LIN {X 0,Y 573.015,Z 252.998,A -85,B 0,C 180,E1 -2072.459,E2 -2072.459} C_VEL
LIN {X 0,Y 573.012,Z 250.251,A -85,B 0,C 180,E1 -2073.163,E2 -2073.163} C_VEL
LIN {X 0,Y 573.036,Z 245.506,A -85,B 0,C 180,E1 -2074.043,E2 -2074.043} C_VEL
LIN {X 0,Y 573.097,Z 240.544,A -85,B 0,C 180,E1 -2074.747,E2 -2074.747} C_VEL
LIN {X 0,Y 573.027,Z 234.186,A -85,B 0,C 180,E1 -2075.453,E2 -2075.453} C_VEL
LIN {X 0,Y 573.106,Z 227.017,A -85,B 0,C 180,E1 -2076.07,E2 -2076.07} C_VEL
LIN {X 0,Y 573.128,Z 220.284,A -85,B 0,C 180,E1 -2076.527,E2 -2076.527} C_VEL
LIN {X 0,Y 573.236,Z 211.927,A -85,B 0,C 180,E1 -2076.962,E2 -2076.962} C_VEL
LIN {X 0,Y 573.056,Z 204.686,A -85,B 0,C 180,E1 -2077.243,E2 -2077.243} C_VEL
LIN {X 0,Y 572.921,Z 203.423,A -85,B 0,C 180,E1 -2077.311,E2 -2077.311} C_VEL
LIN {X 0,Y 572.967,Z 198.327,A -85,B 0,C 180,E1 -2080.601,E2 -2080.601} C_VEL
LIN {X 0,Y 572.969,Z 193.92,A -85,B 0,C 180,E1 -2083.476,E2 -2083.476} C_VEL
LIN {X 0,Y 572.966,Z 189.58,A -85,B 0,C 180,E1 -2086.386,E2 -2086.386} C_VEL
LIN {X 0,Y 572.998,Z 185.595,A -85,B 0,C 180,E1 -2089.338,E2 -2089.338} C_VEL
LIN {X 0,Y 573.019,Z 182.564,A -85,B 0,C 180,E1 -2091.588,E2 -2091.588} C_VEL
LIN {X 0,Y 573.073,Z 179.507,A -85,B 0,C 180,E1 -2093.871,E2 -2093.871} C_VEL
LIN {X 0,Y 573.141,Z 176.057,A -85,B 0,C 180,E1 -2096.472,E2 -2096.472} C_VEL
LIN {X 0,Y 573.16,Z 173.251,A -85,B 0,C 180,E1 -2098.567,E2 -2098.567} C_VEL
LIN {X 0,Y 573.151,Z 172.095,A -85,B 0,C 180,E1 -2099.471,E2 -2099.471} C_VEL
LIN {X 0,Y 573.245,Z 172.076,A -85,B 0,C 180,E1 -2102.227,E2 -2102.227} C_VEL
LIN {X 0,Y 573.233,Z 172.077,A -85,B 0,C 180,E1 -2104.771,E2 -2104.771} C_VEL
LIN {X 0,Y 573.247,Z 172.08,A -85,B 0,C 180,E1 -2107.165,E2 -2107.165} C_VEL
LIN {X 0,Y 573.241,Z 172.079,A -85,B 0,C 180,E1 -2109.606,E2 -2109.606} C_VEL
LIN {X 0,Y 573.237,Z 172.078,A -85,B 0,C 180,E1 -2112.641,E2 -2112.641} C_VEL
LIN {X 0,Y 573.229,Z 172.077,A -85,B 0,C 180,E1 -2115.666,E2 -2115.666} C_VEL
LIN {X 0,Y 573.238,Z 172.08,A -85,B 0,C 180,E1 -2118.543,E2 -2118.543} C_VEL
LIN {X 0,Y 573.242,Z 172.076,A -85,B 0,C 180,E1 -2121.298,E2 -2121.298} C_VEL
LIN {X 0,Y 573.257,Z 172.074,A -85,B 0,C 180,E1 -2124.01,E2 -2124.01} C_VEL
LIN {X 0,Y 573.276,Z 172.079,A -85,B 0,C 180,E1 -2126.518,E2 -2126.518} C_VEL
LIN {X 0,Y 573.236,Z 172.076,A -85,B 0,C 180,E1 -2129.114,E2 -2129.114} C_VEL
LIN {X 0,Y 573.256,Z 172.077,A -85,B 0,C 180,E1 -2131.967,E2 -2131.967} C_VEL
LIN {X 0,Y 573.249,Z 172.075,A -85,B 0,C 180,E1 -2134.59,E2 -2134.59} C_VEL
LIN {X 0,Y 573.23,Z 172.08,A -85,B 0,C 180,E1 -2137.662,E2 -2137.662} C_VEL
LIN {X 0,Y 573.248,Z 172.082,A -85,B 0,C 180,E1 -2139.923,E2 -2139.923} C_VEL
LIN {X 0,Y 573.253,Z 172.074,A -85,B 0,C 180,E1 -2142.988,E2 -2142.988} C_VEL
LIN {X 0,Y 573.263,Z 172.078,A -85,B 0,C 180,E1 -2145.807,E2 -2145.807} C_VEL
LIN {X 0,Y 573.272,Z 172.071,A -85,B 0,C 180,E1 -2148.734,E2 -2148.734} C_VEL
LIN {X 0,Y 573.296,Z 172.074,A -85,B 0,C 180,E1 -2151.541,E2 -2151.541} C_VEL
LIN {X 0,Y 573.283,Z 172.069,A -85,B 0,C 180,E1 -2154.372,E2 -2154.372} C_VEL
LIN {X 0,Y 573.296,Z 172.076,A -85,B 0,C 180,E1 -2157.189,E2 -2157.189} C_VEL
LIN {X 0,Y 573.3,Z 172.066,A -85,B 0,C 180,E1 -2160,E2 -2160} C_VEL
LIN {X 0,Y 573.3,Z 172.076,A -85,B 0,C 180,E1 -2162.811,E2 -2162.811} C_VEL
LIN {X 0,Y 573.265,Z 172.071,A -85,B 0,C 180,E1 -2165.628,E2 -2165.628} C_VEL
LIN {X 0,Y 573.274,Z 172.078,A -85,B 0,C 180,E1 -2168.46,E2 -2168.46} C_VEL
LIN {X 0,Y 573.259,Z 172.073,A -85,B 0,C 180,E1 -2171.312,E2 -2171.312} C_VEL
LIN {X 0,Y 573.268,Z 172.079,A -85,B 0,C 180,E1 -2174.424,E2 -2174.424} C_VEL
LIN {X 0,Y 573.233,Z 172.075,A -85,B 0,C 180,E1 -2177.112,E2 -2177.112} C_VEL
LIN {X 0,Y 573.22,Z 172.087,A -85,B 0,C 180,E1 -2180.078,E2 -2180.078} C_VEL
LIN {X 0,Y 573.204,Z 172.083,A -85,B 0,C 180,E1 -2182.339,E2 -2182.339} C_VEL
LIN {X 0,Y 573.212,Z 172.082,A -85,B 0,C 180,E1 -2185.412,E2 -2185.412} C_VEL
LIN {X 0,Y 573.166,Z 172.084,A -85,B 0,C 180,E1 -2188.568,E2 -2188.568} C_VEL
LIN {X 0,Y 573.204,Z 172.081,A -85,B 0,C 180,E1 -2190.995,E2 -2190.995} C_VEL
LIN {X 0,Y 573.253,Z 172.081,A -85,B 0,C 180,E1 -2193.525,E2 -2193.525} C_VEL
LIN {X 0,Y 573.177,Z 172.084,A -85,B 0,C 180,E1 -2196.054,E2 -2196.054} C_VEL
LIN {X 0,Y 573.225,Z 172.08,A -85,B 0,C 180,E1 -2198.703,E2 -2198.703} C_VEL
LIN {X 0,Y 573.205,Z 172.082,A -85,B 0,C 180,E1 -2201.592,E2 -2201.592} C_VEL
LIN {X 0,Y 573.214,Z 172.08,A -85,B 0,C 180,E1 -2204.336,E2 -2204.336} C_VEL
LIN {X 0,Y 573.233,Z 172.076,A -85,B 0,C 180,E1 -2207.36,E2 -2207.36} C_VEL
LIN {X 0,Y 573.239,Z 172.081,A -85,B 0,C 180,E1 -2210.394,E2 -2210.394} C_VEL
LIN {X 0,Y 573.247,Z 172.077,A -85,B 0,C 180,E1 -2213.079,E2 -2213.079} C_VEL
LIN {X 0,Y 573.262,Z 172.073,A -85,B 0,C 180,E1 -2215.672,E2 -2215.672} C_VEL
LIN {X 0,Y 573.241,Z 172.084,A -85,B 0,C 180,E1 -2218.186,E2 -2218.186} C_VEL
LIN {X 0,Y 573.246,Z 172.092,A -85,B 0,C 180,E1 -2219.909,E2 -2219.909} C_VEL
LIN {X 0,Y 574.683,Z 179.226,A -85,B 0,C 180,E1 -2221.116,E2 -2221.116} C_VEL
LIN {X 0,Y 574.417,Z 195.626,A -85,B 0,C 180,E1 -2223.566,E2 -2223.566} C_VEL
LIN {X 0,Y 574.13,Z 214.897,A -85,B 0,C 180,E1 -2226.339,E2 -2226.339} C_VEL
LIN {X 0,Y 573.948,Z 232.888,A -85,B 0,C 180,E1 -2228.868,E2 -2228.868} C_VEL
LIN {X 0,Y 573.731,Z 253.864,A -85,B 0,C 180,E1 -2231.799,E2 -2231.799} C_VEL
LIN {X 0,Y 573.504,Z 273.808,A -85,B 0,C 180,E1 -2234.543,E2 -2234.543} C_VEL
LIN {X 0,Y 573.35,Z 293.752,A -85,B 0,C 180,E1 -2237.254,E2 -2237.254} C_VEL
LIN {X 0,Y 573.34,Z 295.393,A -85,B 0,C 180,E1 -2237.434,E2 -2237.434} C_VEL
LIN {X 0,Y 573.925,Z 301.68,A -85,B 0,C 180,E1 -2237.537,E2 -2237.537} C_VEL
LIN {X 0,Y 573.782,Z 314.725,A -85,B 0,C 180,E1 -2237.826,E2 -2237.826} C_VEL
LIN {X 0,Y 573.709,Z 327.272,A -85,B 0,C 180,E1 -2238.25,E2 -2238.25} C_VEL
LIN {X 0,Y 573.61,Z 338.953,A -85,B 0,C 180,E1 -2238.785,E2 -2238.785} C_VEL
LIN {X 0,Y 573.478,Z 349.603,A -85,B 0,C 180,E1 -2239.408,E2 -2239.408} C_VEL
LIN {X 0,Y 573.362,Z 360.484,A -85,B 0,C 180,E1 -2240.209,E2 -2240.209} C_VEL
LIN {X 0,Y 573.24,Z 371.123,A -85,B 0,C 180,E1 -2241.186,E2 -2241.186} C_VEL
LIN {X 0,Y 573.16,Z 378.968,A -85,B 0,C 180,E1 -2242.072,E2 -2242.072} C_VEL
LIN {X 0,Y 573.073,Z 386.586,A -85,B 0,C 180,E1 -2243.127,E2 -2243.127} C_VEL
LIN {X 0,Y 573.07,Z 393.684,A -85,B 0,C 180,E1 -2244.371,E2 -2244.371} C_VEL
LIN {X 0,Y 573.028,Z 398.375,A -85,B 0,C 180,E1 -2245.428,E2 -2245.428} C_VEL
LIN {X 0,Y 573.022,Z 401.962,A -85,B 0,C 180,E1 -2246.485,E2 -2246.485} C_VEL
LIN {X 0,Y 572.959,Z 403.812,A -85,B 0,C 180,E1 -2247.189,E2 -2247.189} C_VEL
LIN {X 0,Y 572.94,Z 405.201,A -85,B 0,C 180,E1 -2247.892,E2 -2247.892} C_VEL
LIN {X 0,Y 572.94,Z 406.786,A -85,B 0,C 180,E1 -2249.298,E2 -2249.298} C_VEL
LIN {X 0,Y 572.938,Z 407,A -85,B 0,C 180,E1 -2250.001,E2 -2250.001} C_VEL
LIN {X 0,Y 572.946,Z 406.185,A -85,B 0,C 180,E1 -2251.407,E2 -2251.407} C_VEL
LIN {X 0,Y 572.94,Z 405.197,A -85,B 0,C 180,E1 -2252.11,E2 -2252.11} C_VEL
LIN {X 0,Y 572.959,Z 403.806,A -85,B 0,C 180,E1 -2252.813,E2 -2252.813} C_VEL
LIN {X 0,Y 573.015,Z 400.893,A -85,B 0,C 180,E1 -2253.869,E2 -2253.869} C_VEL
LIN {X 0,Y 572.963,Z 396.946,A -85,B 0,C 180,E1 -2254.926,E2 -2254.926} C_VEL
LIN {X 0,Y 573.065,Z 390.872,A -85,B 0,C 180,E1 -2256.161,E2 -2256.161} C_VEL
LIN {X 0,Y 573.12,Z 384.232,A -85,B 0,C 180,E1 -2257.222,E2 -2257.222} C_VEL
LIN {X 0,Y 573.199,Z 375.984,A -85,B 0,C 180,E1 -2258.284,E2 -2258.284} C_VEL
LIN {X 0,Y 573.287,Z 367.53,A -85,B 0,C 180,E1 -2259.171,E2 -2259.171} C_VEL
LIN {X 0,Y 573.426,Z 357.088,A -85,B 0,C 180,E1 -2260.059,E2 -2260.059} C_VEL
LIN {X 0,Y 573.537,Z 345.389,A -85,B 0,C 180,E1 -2260.856,E2 -2260.856} C_VEL
LIN {X 0,Y 573.654,Z 334.274,A -85,B 0,C 180,E1 -2261.448,E2 -2261.448} C_VEL
LIN {X 0,Y 573.759,Z 321.154,A -85,B 0,C 180,E1 -2261.975,E2 -2261.975} C_VEL
LIN {X 0,Y 573.845,Z 308.489,A -85,B 0,C 180,E1 -2262.332,E2 -2262.332} C_VEL
LIN {X 0,Y 573.821,Z 298.547,A -85,B 0,C 180,E1 -2262.512,E2 -2262.512} C_VEL
LIN {X 0,Y 573.297,Z 294.902,A -85,B 0,C 180,E1 -2262.591,E2 -2262.591} C_VEL
LIN {X 0,Y 573.449,Z 276.454,A -85,B 0,C 180,E1 -2265.097,E2 -2265.097} C_VEL
LIN {X 0,Y 573.671,Z 256.51,A -85,B 0,C 180,E1 -2267.836,E2 -2267.836} C_VEL
LIN {X 0,Y 573.902,Z 236.566,A -85,B 0,C 180,E1 -2270.615,E2 -2270.615} C_VEL
LIN {X 0,Y 574.126,Z 217.882,A -85,B 0,C 180,E1 -2273.24,E2 -2273.24} C_VEL
LIN {X 0,Y 574.361,Z 197.613,A -85,B 0,C 180,E1 -2276.137,E2 -2276.137} C_VEL
LIN {X 0,Y 574.695,Z 180.513,A -85,B 0,C 180,E1 -2278.686,E2 -2278.686} C_VEL
LIN {X 0,Y 574.272,Z 176.66,A -85,B 0,C 180,E1 -2279.31,E2 -2279.31} C_VEL
LIN {X 0,Y 573.228,Z 172.084,A -85,B 0,C 180,E1 -2280.094,E2 -2280.094} C_VEL
LIN {X 0,Y 573.226,Z 172.082,A -85,B 0,C 180,E1 -2282.648,E2 -2282.648} C_VEL
LIN {X 0,Y 573.191,Z 172.089,A -85,B 0,C 180,E1 -2285.19,E2 -2285.19} C_VEL
LIN {X 0,Y 573.231,Z 172.079,A -85,B 0,C 180,E1 -2287.809,E2 -2287.809} C_VEL
LIN {X 0,Y 573.25,Z 172.08,A -85,B 0,C 180,E1 -2290.525,E2 -2290.525} C_VEL
LIN {X 0,Y 573.241,Z 172.078,A -85,B 0,C 180,E1 -2293.36,E2 -2293.36} C_VEL
LIN {X 0,Y 573.241,Z 172.077,A -85,B 0,C 180,E1 -2296.641,E2 -2296.641} C_VEL
LIN {X 0,Y 573.25,Z 172.08,A -85,B 0,C 180,E1 -2299.475,E2 -2299.475} C_VEL
LIN {X 0,Y 573.229,Z 172.08,A -85,B 0,C 180,E1 -2302.192,E2 -2302.192} C_VEL
LIN {X 0,Y 573.205,Z 172.084,A -85,B 0,C 180,E1 -2305.234,E2 -2305.234} C_VEL
LIN {X 0,Y 573.152,Z 172.129,A -85,B 0,C 180,E1 -2306.088,E2 -2306.088} C_VEL
LIN {X 0,Y 573.182,Z 181.357,A -85,B 0,C 180,E1 -2308.593,E2 -2308.593} C_VEL
LIN {X 0,Y 573.206,Z 191.116,A -85,B 0,C 180,E1 -2311.434,E2 -2311.434} C_VEL
LIN {X 0,Y 573.264,Z 200.054,A -85,B 0,C 180,E1 -2314.201,E2 -2314.201} C_VEL
LIN {X 0,Y 573.203,Z 208.222,A -85,B 0,C 180,E1 -2316.899,E2 -2316.899} C_VEL
LIN {X 0,Y 573.192,Z 215.13,A -85,B 0,C 180,E1 -2319.171,E2 -2319.171} C_VEL
LIN {X 0,Y 573.142,Z 222.895,A -85,B 0,C 180,E1 -2321.779,E2 -2321.779} C_VEL
LIN {X 0,Y 573.106,Z 230.685,A -85,B 0,C 180,E1 -2324.348,E2 -2324.348} C_VEL
LIN {X 0,Y 573.075,Z 239.587,A -85,B 0,C 180,E1 -2327.247,E2 -2327.247} C_VEL
LIN {X 0,Y 573.088,Z 240.711,A -85,B 0,C 180,E1 -2327.551,E2 -2327.551} C_VEL
LIN {X 0,Y 573.868,Z 246.446,A -85,B 0,C 180,E1 -2327.669,E2 -2327.669} C_VEL
LIN {X 0,Y 573.774,Z 259.872,A -85,B 0,C 180,E1 -2328.026,E2 -2328.026} C_VEL
LIN {X 0,Y 573.64,Z 271.829,A -85,B 0,C 180,E1 -2328.485,E2 -2328.485} C_VEL
LIN {X 0,Y 573.551,Z 283.172,A -85,B 0,C 180,E1 -2329.061,E2 -2329.061} C_VEL
LIN {X 0,Y 573.454,Z 294.108,A -85,B 0,C 180,E1 -2329.764,E2 -2329.764} C_VEL
LIN {X 0,Y 573.34,Z 303.126,A -85,B 0,C 180,E1 -2330.475,E2 -2330.475} C_VEL
LIN {X 0,Y 573.244,Z 312.371,A -85,B 0,C 180,E1 -2331.362,E2 -2331.362} C_VEL
LIN {X 0,Y 573.143,Z 321.354,A -85,B 0,C 180,E1 -2332.425,E2 -2332.425} C_VEL
LIN {X 0,Y 573.091,Z 327.919,A -85,B 0,C 180,E1 -2333.382,E2 -2333.382} C_VEL
LIN {X 0,Y 573.071,Z 333.463,A -85,B 0,C 180,E1 -2334.37,E2 -2334.37} C_VEL
LIN {X 0,Y 573.029,Z 338.204,A -85,B 0,C 180,E1 -2335.428,E2 -2335.428} C_VEL
LIN {X 0,Y 573.022,Z 341.832,A -85,B 0,C 180,E1 -2336.484,E2 -2336.484} C_VEL
LIN {X 0,Y 572.959,Z 343.69,A -85,B 0,C 180,E1 -2337.188,E2 -2337.188} C_VEL
LIN {X 0,Y 572.938,Z 345.134,A -85,B 0,C 180,E1 -2337.891,E2 -2337.891} C_VEL
LIN {X 0,Y 572.942,Z 346.754,A -85,B 0,C 180,E1 -2339.297,E2 -2339.297} C_VEL
LIN {X 0,Y 572.938,Z 346.996,A -85,B 0,C 180,E1 -2340,E2 -2340} C_VEL
LIN {X 0,Y 572.941,Z 346.813,A -85,B 0,C 180,E1 -2340.703,E2 -2340.703} C_VEL
LIN {X 0,Y 572.937,Z 345.275,A -85,B 0,C 180,E1 -2342.109,E2 -2342.109} C_VEL
LIN {X 0,Y 572.96,Z 343.908,A -85,B 0,C 180,E1 -2342.812,E2 -2342.812} C_VEL
LIN {X 0,Y 573.015,Z 341.039,A -85,B 0,C 180,E1 -2343.868,E2 -2343.868} C_VEL
LIN {X 0,Y 572.963,Z 337.14,A -85,B 0,C 180,E1 -2344.926,E2 -2344.926} C_VEL
LIN {X 0,Y 573.075,Z 332.097,A -85,B 0,C 180,E1 -2345.984,E2 -2345.984} C_VEL
LIN {X 0,Y 573.084,Z 325.762,A -85,B 0,C 180,E1 -2347.044,E2 -2347.044} C_VEL
LIN {X 0,Y 573.175,Z 317.867,A -85,B 0,C 180,E1 -2348.106,E2 -2348.106} C_VEL
LIN {X 0,Y 573.254,Z 309.793,A -85,B 0,C 180,E1 -2348.993,E2 -2348.993} C_VEL
LIN {X 0,Y 573.336,Z 299.936,A -85,B 0,C 180,E1 -2349.882,E2 -2349.882} C_VEL
LIN {X 0,Y 573.464,Z 288.94,A -85,B 0,C 180,E1 -2350.679,E2 -2350.679} C_VEL
LIN {X 0,Y 573.587,Z 276.923,A -85,B 0,C 180,E1 -2351.364,E2 -2351.364} C_VEL
LIN {X 0,Y 573.702,Z 264.987,A -85,B 0,C 180,E1 -2351.886,E2 -2351.886} C_VEL
LIN {X 0,Y 573.833,Z 251.33,A -85,B 0,C 180,E1 -2352.309,E2 -2352.309} C_VEL
LIN {X 0,Y 573.604,Z 244.173,A -85,B 0,C 180,E1 -2352.471,E2 -2352.471} C_VEL
LIN {X 0,Y 573.043,Z 240.491,A -85,B 0,C 180,E1 -2352.551,E2 -2352.551} C_VEL
LIN {X 0,Y 573.085,Z 230.959,A -85,B 0,C 180,E1 -2355.652,E2 -2355.652} C_VEL
LIN {X 0,Y 573.102,Z 223.166,A -85,B 0,C 180,E1 -2358.223,E2 -2358.223} C_VEL
LIN {X 0,Y 573.143,Z 221.241,A -85,B 0,C 180,E1 -2358.862,E2 -2358.862} C_VEL
LIN {X 0,Y 572.509,Z 219.635,A -85,B 0,C 180,E1 -2359.426,E2 -2359.426} C_VEL
LIN {X 0,Y 569.679,Z 217.271,A -85,B 0,C 180,E1 -2360.35,E2 -2360.35} C_VEL
LIN {X 0,Y 567.27,Z 215.411,A -85,B 0,C 180,E1 -2361.093,E2 -2361.093} C_VEL
LIN {X 0,Y 566.231,Z 213.9,A -85,B 0,C 180,E1 -2361.665,E2 -2361.665} C_VEL
LIN {X 0,Y 566.145,Z 213.329,A -85,B 0,C 180,E1 -2361.857,E2 -2361.857} C_VEL
LIN {X 0,Y 566.188,Z 205.251,A -85,B 0,C 180,E1 -2364.572,E2 -2364.572} C_VEL
LIN {X 0,Y 566.243,Z 197.135,A -85,B 0,C 180,E1 -2367.338,E2 -2367.338} C_VEL
LIN {X 0,Y 566.283,Z 189.921,A -85,B 0,C 180,E1 -2369.764,E2 -2369.764} C_VEL
LIN {X 0,Y 566.353,Z 182.564,A -85,B 0,C 180,E1 -2372.249,E2 -2372.249} C_VEL
LIN {X 0,Y 566.349,Z 174.409,A -85,B 0,C 180,E1 -2375.013,E2 -2375.013} C_VEL
LIN {X 0,Y 566.156,Z 172.965,A -85,B 0,C 180,E1 -2375.555,E2 -2375.555} C_VEL
LIN {X 0,Y 566.211,Z 172.954,A -85,B 0,C 180,E1 -2378.557,E2 -2378.557} C_VEL
LIN {X 0,Y 566.177,Z 172.964,A -85,B 0,C 180,E1 -2381.14,E2 -2381.14} C_VEL
LIN {X 0,Y 566.162,Z 172.961,A -85,B 0,C 180,E1 -2383.947,E2 -2383.947} C_VEL
LIN {X 0,Y 566.205,Z 172.955,A -85,B 0,C 180,E1 -2386.945,E2 -2386.945} C_VEL
LIN {X 0,Y 566.212,Z 172.953,A -85,B 0,C 180,E1 -2389.801,E2 -2389.801} C_VEL
LIN {X 0,Y 566.191,Z 172.959,A -85,B 0,C 180,E1 -2392.601,E2 -2392.601} C_VEL
LIN {X 0,Y 566.189,Z 172.959,A -85,B 0,C 180,E1 -2395.18,E2 -2395.18} C_VEL
LIN {X 0,Y 566.235,Z 172.951,A -85,B 0,C 180,E1 -2397.743,E2 -2397.743} C_VEL
LIN {X 0,Y 566.122,Z 172.971,A -85,B 0,C 180,E1 -2400.343,E2 -2400.343} C_VEL
LIN {X 0,Y 566.099,Z 173.398,A -85,B 0,C 180,E1 -2401.041,E2 -2401.041} C_VEL
LIN {X 0,Y 566.102,Z 176.607,A -85,B 0,C 180,E1 -2403.452,E2 -2403.452} C_VEL
LIN {X 0,Y 566.036,Z 179.691,A -85,B 0,C 180,E1 -2405.811,E2 -2405.811} C_VEL
LIN {X 0,Y 565.978,Z 183.82,A -85,B 0,C 180,E1 -2408.893,E2 -2408.893} C_VEL
LIN {X 0,Y 565.914,Z 187.813,A -85,B 0,C 180,E1 -2411.912,E2 -2411.912} C_VEL
LIN {X 0,Y 565.885,Z 190.906,A -85,B 0,C 180,E1 -2414.143,E2 -2414.143} C_VEL
LIN {X 0,Y 565.881,Z 193.87,A -85,B 0,C 180,E1 -2416.35,E2 -2416.35} C_VEL
LIN {X 0,Y 565.884,Z 198.186,A -85,B 0,C 180,E1 -2419.263,E2 -2419.263} C_VEL
LIN {X 0,Y 565.857,Z 203.453,A -85,B 0,C 180,E1 -2422.708,E2 -2422.708} C_VEL
LIN {X 0,Y 566.167,Z 211.205,A -85,B 0,C 180,E1 -2423.01,E2 -2423.01} C_VEL
LIN {X 0,Y 566.114,Z 218.9,A -85,B 0,C 180,E1 -2423.401,E2 -2423.401} C_VEL
LIN {X 0,Y 566.062,Z 225.793,A -85,B 0,C 180,E1 -2423.852,E2 -2423.852} C_VEL
LIN {X 0,Y 565.983,Z 231.354,A -85,B 0,C 180,E1 -2424.298,E2 -2424.298} C_VEL
LIN {X 0,Y 566.01,Z 238.313,A -85,B 0,C 180,E1 -2425.013,E2 -2425.013} C_VEL
LIN {X 0,Y 565.97,Z 243.753,A -85,B 0,C 180,E1 -2425.726,E2 -2425.726} C_VEL
LIN {X 0,Y 565.969,Z 248.043,A -85,B 0,C 180,E1 -2426.439,E2 -2426.439} C_VEL
LIN {X 0,Y 565.892,Z 251.374,A -85,B 0,C 180,E1 -2427.152,E2 -2427.152} C_VEL
LIN {X 0,Y 565.855,Z 253.859,A -85,B 0,C 180,E1 -2427.864,E2 -2427.864} C_VEL
LIN {X 0,Y 565.847,Z 255.567,A -85,B 0,C 180,E1 -2428.576,E2 -2428.576} C_VEL
LIN {X 0,Y 565.841,Z 256.57,A -85,B 0,C 180,E1 -2429.287,E2 -2429.287} C_VEL
LIN {X 0,Y 565.839,Z 256.937,A -85,B 0,C 180,E1 -2429.999,E2 -2429.999} C_VEL
LIN {X 0,Y 565.841,Z 256.676,A -85,B 0,C 180,E1 -2430.711,E2 -2430.711} C_VEL
LIN {X 0,Y 565.848,Z 255.761,A -85,B 0,C 180,E1 -2431.422,E2 -2431.422} C_VEL
LIN {X 0,Y 565.854,Z 254.12,A -85,B 0,C 180,E1 -2432.134,E2 -2432.134} C_VEL
LIN {X 0,Y 565.935,Z 250.247,A -85,B 0,C 180,E1 -2433.203,E2 -2433.203} C_VEL
LIN {X 0,Y 565.952,Z 245.495,A -85,B 0,C 180,E1 -2434.094,E2 -2434.094} C_VEL
LIN {X 0,Y 566.024,Z 240.534,A -85,B 0,C 180,E1 -2434.807,E2 -2434.807} C_VEL
LIN {X 0,Y 565.954,Z 234.166,A -85,B 0,C 180,E1 -2435.522,E2 -2435.522} C_VEL
LIN {X 0,Y 566.045,Z 228.167,A -85,B 0,C 180,E1 -2436.057,E2 -2436.057} C_VEL
LIN {X 0,Y 566.071,Z 220.396,A -85,B 0,C 180,E1 -2436.601,E2 -2436.601} C_VEL
LIN {X 0,Y 566.152,Z 214.044,A -85,B 0,C 180,E1 -2436.953,E2 -2436.953} C_VEL
LIN {X 0,Y 566.153,Z 206.734,A -85,B 0,C 180,E1 -2437.264,E2 -2437.264} C_VEL
LIN {X 0,Y 565.854,Z 203.456,A -85,B 0,C 180,E1 -2437.38,E2 -2437.38} C_VEL
LIN {X 0,Y 565.879,Z 198.326,A -85,B 0,C 180,E1 -2440.736,E2 -2440.736} C_VEL
LIN {X 0,Y 565.871,Z 193.997,A -85,B 0,C 180,E1 -2443.648,E2 -2443.648} C_VEL
LIN {X 0,Y 565.916,Z 190.002,A -85,B 0,C 180,E1 -2446.596,E2 -2446.596} C_VEL
LIN {X 0,Y 565.936,Z 185.968,A -85,B 0,C 180,E1 -2449.589,E2 -2449.589} C_VEL
LIN {X 0,Y 565.963,Z 182.909,A -85,B 0,C 180,E1 -2451.871,E2 -2451.871} C_VEL
LIN {X 0,Y 566.03,Z 179.83,A -85,B 0,C 180,E1 -2454.187,E2 -2454.187} C_VEL
LIN {X 0,Y 566.079,Z 176.631,A -85,B 0,C 180,E1 -2456.633,E2 -2456.633} C_VEL
LIN {X 0,Y 566.102,Z 173.527,A -85,B 0,C 180,E1 -2458.957,E2 -2458.957} C_VEL
LIN {X 0,Y 566.126,Z 172.97,A -85,B 0,C 180,E1 -2459.772,E2 -2459.772} C_VEL
LIN {X 0,Y 566.198,Z 172.953,A -85,B 0,C 180,E1 -2462.428,E2 -2462.428} C_VEL
LIN {X 0,Y 566.195,Z 172.955,A -85,B 0,C 180,E1 -2464.991,E2 -2464.991} C_VEL
LIN {X 0,Y 566.191,Z 172.961,A -85,B 0,C 180,E1 -2467.46,E2 -2467.46} C_VEL
LIN {X 0,Y 566.212,Z 172.95,A -85,B 0,C 180,E1 -2470.197,E2 -2470.197} C_VEL
LIN {X 0,Y 566.199,Z 172.96,A -85,B 0,C 180,E1 -2473.053,E2 -2473.053} C_VEL
LIN {X 0,Y 566.193,Z 172.953,A -85,B 0,C 180,E1 -2476.047,E2 -2476.047} C_VEL
LIN {X 0,Y 566.205,Z 172.96,A -85,B 0,C 180,E1 -2478.863,E2 -2478.863} C_VEL
LIN {X 0,Y 566.182,Z 172.954,A -85,B 0,C 180,E1 -2481.636,E2 -2481.636} C_VEL
LIN {X 0,Y 566.205,Z 172.956,A -85,B 0,C 180,E1 -2484.311,E2 -2484.311} C_VEL
LIN {X 0,Y 566.221,Z 172.952,A -85,B 0,C 180,E1 -2486.898,E2 -2486.898} C_VEL
LIN {X 0,Y 566.185,Z 172.953,A -85,B 0,C 180,E1 -2489.407,E2 -2489.407} C_VEL
LIN {X 0,Y 566.219,Z 172.952,A -85,B 0,C 180,E1 -2491.858,E2 -2491.858} C_VEL
LIN {X 0,Y 566.217,Z 172.956,A -85,B 0,C 180,E1 -2494.251,E2 -2494.251} C_VEL
LIN {X 0,Y 566.183,Z 172.955,A -85,B 0,C 180,E1 -2496.713,E2 -2496.713} C_VEL
LIN {X 0,Y 566.21,Z 172.955,A -85,B 0,C 180,E1 -2499.663,E2 -2499.663} C_VEL
LIN {X 0,Y 566.194,Z 172.953,A -85,B 0,C 180,E1 -2502.668,E2 -2502.668} C_VEL
LIN {X 0,Y 566.223,Z 172.956,A -85,B 0,C 180,E1 -2505.626,E2 -2505.626} C_VEL
LIN {X 0,Y 566.264,Z 172.944,A -85,B 0,C 180,E1 -2508.654,E2 -2508.654} C_VEL
LIN {X 0,Y 566.238,Z 172.955,A -85,B 0,C 180,E1 -2511.434,E2 -2511.434} C_VEL
LIN {X 0,Y 566.249,Z 172.945,A -85,B 0,C 180,E1 -2514.302,E2 -2514.302} C_VEL
LIN {X 0,Y 566.26,Z 172.944,A -85,B 0,C 180,E1 -2517.866,E2 -2517.866} C_VEL
LIN {X 0,Y 566.299,Z 172.943,A -85,B 0,C 180,E1 -2520.711,E2 -2520.711} C_VEL
LIN {X 0,Y 566.265,Z 172.953,A -85,B 0,C 180,E1 -2522.846,E2 -2522.846} C_VEL
LIN {X 0,Y 566.234,Z 172.947,A -85,B 0,C 180,E1 -2525.699,E2 -2525.699} C_VEL
LIN {X 0,Y 566.217,Z 172.958,A -85,B 0,C 180,E1 -2528.566,E2 -2528.566} C_VEL
LIN {X 0,Y 566.229,Z 172.948,A -85,B 0,C 180,E1 -2531.455,E2 -2531.455} C_VEL
LIN {X 0,Y 566.221,Z 172.956,A -85,B 0,C 180,E1 -2534.506,E2 -2534.506} C_VEL
LIN {X 0,Y 566.175,Z 172.954,A -85,B 0,C 180,E1 -2537.332,E2 -2537.332} C_VEL
LIN {X 0,Y 566.186,Z 172.956,A -85,B 0,C 180,E1 -2539.582,E2 -2539.582} C_VEL
LIN {X 0,Y 566.171,Z 172.964,A -85,B 0,C 180,E1 -2541.864,E2 -2541.864} C_VEL
LIN {X 0,Y 566.166,Z 172.957,A -85,B 0,C 180,E1 -2545.022,E2 -2545.022} C_VEL
LIN {X 0,Y 566.145,Z 172.963,A -85,B 0,C 180,E1 -2547.343,E2 -2547.343} C_VEL
LIN {X 0,Y 566.147,Z 172.965,A -85,B 0,C 180,E1 -2549.772,E2 -2549.772} C_VEL
LIN {X 0,Y 566.181,Z 172.954,A -85,B 0,C 180,E1 -2552.429,E2 -2552.429} C_VEL
LIN {X 0,Y 566.158,Z 172.96,A -85,B 0,C 180,E1 -2554.989,E2 -2554.989} C_VEL
LIN {X 0,Y 566.181,Z 172.961,A -85,B 0,C 180,E1 -2557.462,E2 -2557.462} C_VEL
LIN {X 0,Y 566.196,Z 172.951,A -85,B 0,C 180,E1 -2560.2,E2 -2560.2} C_VEL
LIN {X 0,Y 566.186,Z 172.962,A -85,B 0,C 180,E1 -2563.056,E2 -2563.056} C_VEL
LIN {X 0,Y 566.186,Z 172.954,A -85,B 0,C 180,E1 -2566.05,E2 -2566.05} C_VEL
LIN {X 0,Y 566.197,Z 172.956,A -85,B 0,C 180,E1 -2569.216,E2 -2569.216} C_VEL
LIN {X 0,Y 566.179,Z 172.956,A -85,B 0,C 180,E1 -2571.638,E2 -2571.638} C_VEL
LIN {X 0,Y 566.159,Z 172.964,A -85,B 0,C 180,E1 -2574.309,E2 -2574.309} C_VEL
LIN {X 0,Y 566.216,Z 172.955,A -85,B 0,C 180,E1 -2576.899,E2 -2576.899} C_VEL
LIN {X 0,Y 566.195,Z 172.997,A -85,B 0,C 180,E1 -2579.668,E2 -2579.668} C_VEL
LIN {X 0,Y 567.802,Z 180.39,A -85,B 0,C 180,E1 -2580.935,E2 -2580.935} C_VEL
LIN {X 0,Y 567.543,Z 195.923,A -85,B 0,C 180,E1 -2583.296,E2 -2583.296} C_VEL
LIN {X 0,Y 567.281,Z 213.486,A -85,B 0,C 180,E1 -2585.87,E2 -2585.87} C_VEL
LIN {X 0,Y 567.038,Z 233.068,A -85,B 0,C 180,E1 -2588.652,E2 -2588.652} C_VEL
LIN {X 0,Y 566.762,Z 252.535,A -85,B 0,C 180,E1 -2591.38,E2 -2591.38} C_VEL
LIN {X 0,Y 566.546,Z 271.149,A -85,B 0,C 180,E1 -2593.979,E2 -2593.979} C_VEL
LIN {X 0,Y 566.333,Z 291.093,A -85,B 0,C 180,E1 -2596.729,E2 -2596.729} C_VEL
LIN {X 0,Y 566.302,Z 294.915,A -85,B 0,C 180,E1 -2597.253,E2 -2597.253} C_VEL
LIN {X 0,Y 567.001,Z 301.679,A -85,B 0,C 180,E1 -2597.382,E2 -2597.382} C_VEL
LIN {X 0,Y 566.846,Z 314.723,A -85,B 0,C 180,E1 -2597.674,E2 -2597.674} C_VEL
LIN {X 0,Y 566.745,Z 328.397,A -85,B 0,C 180,E1 -2598.149,E2 -2598.149} C_VEL
LIN {X 0,Y 566.627,Z 340.071,A -85,B 0,C 180,E1 -2598.704,E2 -2598.704} C_VEL
LIN {X 0,Y 566.477,Z 350.923,A -85,B 0,C 180,E1 -2599.366,E2 -2599.366} C_VEL
LIN {X 0,Y 566.335,Z 361.551,A -85,B 0,C 180,E1 -2600.176,E2 -2600.176} C_VEL
LIN {X 0,Y 566.206,Z 371.123,A -85,B 0,C 180,E1 -2601.075,E2 -2601.075} C_VEL
LIN {X 0,Y 566.111,Z 378.968,A -85,B 0,C 180,E1 -2601.973,E2 -2601.973} C_VEL
LIN {X 0,Y 566,Z 386.629,A -85,B 0,C 180,E1 -2603.048,E2 -2603.048} C_VEL
LIN {X 0,Y 566.004,Z 393.684,A -85,B 0,C 180,E1 -2604.3,E2 -2604.3} C_VEL
LIN {X 0,Y 565.933,Z 398.375,A -85,B 0,C 180,E1 -2605.371,E2 -2605.371} C_VEL
LIN {X 0,Y 565.927,Z 401.962,A -85,B 0,C 180,E1 -2606.441,E2 -2606.441} C_VEL
LIN {X 0,Y 565.878,Z 403.812,A -85,B 0,C 180,E1 -2607.153,E2 -2607.153} C_VEL
LIN {X 0,Y 565.846,Z 406.187,A -85,B 0,C 180,E1 -2608.578,E2 -2608.578} C_VEL
LIN {X 0,Y 565.839,Z 407,A -85,B 0,C 180,E1 -2610.001,E2 -2610.001} C_VEL
LIN {X 0,Y 565.846,Z 406.184,A -85,B 0,C 180,E1 -2611.424,E2 -2611.424} C_VEL
LIN {X 0,Y 565.878,Z 403.806,A -85,B 0,C 180,E1 -2612.848,E2 -2612.848} C_VEL
LIN {X 0,Y 565.926,Z 400.892,A -85,B 0,C 180,E1 -2613.917,E2 -2613.917} C_VEL
LIN {X 0,Y 565.878,Z 396.946,A -85,B 0,C 180,E1 -2614.988,E2 -2614.988} C_VEL
LIN {X 0,Y 566.002,Z 391.863,A -85,B 0,C 180,E1 -2616.059,E2 -2616.059} C_VEL
LIN {X 0,Y 566.041,Z 385.462,A -85,B 0,C 180,E1 -2617.133,E2 -2617.133} C_VEL
LIN {X 0,Y 566.133,Z 377.471,A -85,B 0,C 180,E1 -2618.209,E2 -2618.209} C_VEL
LIN {X 0,Y 566.229,Z 369.326,A -85,B 0,C 180,E1 -2619.106,E2 -2619.106} C_VEL
LIN {X 0,Y 566.346,Z 359.391,A -85,B 0,C 180,E1 -2620.006,E2 -2620.006} C_VEL
LIN {X 0,Y 566.53,Z 348.289,A -85,B 0,C 180,E1 -2620.807,E2 -2620.807} C_VEL
LIN {X 0,Y 566.614,Z 337.159,A -85,B 0,C 180,E1 -2621.448,E2 -2621.448} C_VEL
LIN {X 0,Y 566.744,Z 324.968,A -85,B 0,C 180,E1 -2621.989,E2 -2621.989} C_VEL
LIN {X 0,Y 566.859,Z 312.149,A -85,B 0,C 180,E1 -2622.395,E2 -2622.395} C_VEL
LIN {X 0,Y 566.828,Z 298.865,A -85,B 0,C 180,E1 -2622.664,E2 -2622.664} C_VEL
LIN {X 0,Y 566.304,Z 294.902,A -85,B 0,C 180,E1 -2622.749,E2 -2622.749} C_VEL
LIN {X 0,Y 566.453,Z 276.453,A -85,B 0,C 180,E1 -2625.288,E2 -2625.288} C_VEL
LIN {X 0,Y 566.707,Z 257.839,A -85,B 0,C 180,E1 -2627.875,E2 -2627.875} C_VEL
LIN {X 0,Y 566.97,Z 237.845,A -85,B 0,C 180,E1 -2630.689,E2 -2630.689} C_VEL
LIN {X 0,Y 567.198,Z 217.73,A -85,B 0,C 180,E1 -2633.521,E2 -2633.521} C_VEL
LIN {X 0,Y 567.504,Z 198.775,A -85,B 0,C 180,E1 -2636.279,E2 -2636.279} C_VEL
LIN {X 0,Y 567.866,Z 181.654,A -85,B 0,C 180,E1 -2638.861,E2 -2638.861} C_VEL
LIN {X 0,Y 566.907,Z 176.128,A -85,B 0,C 180,E1 -2639.796,E2 -2639.796} C_VEL
LIN {X 0,Y 566.204,Z 172.958,A -85,B 0,C 180,E1 -2640.386,E2 -2640.386} C_VEL
LIN {X 0,Y 566.166,Z 172.966,A -85,B 0,C 180,E1 -2643.106,E2 -2643.106} C_VEL
LIN {X 0,Y 566.144,Z 172.963,A -85,B 0,C 180,E1 -2645.694,E2 -2645.694} C_VEL
LIN {X 0,Y 566.209,Z 172.96,A -85,B 0,C 180,E1 -2648.558,E2 -2648.558} C_VEL
LIN {X 0,Y 566.177,Z 172.956,A -85,B 0,C 180,E1 -2651.14,E2 -2651.14} C_VEL
LIN {X 0,Y 566.196,Z 172.959,A -85,B 0,C 180,E1 -2654.037,E2 -2654.037} C_VEL
LIN {X 0,Y 566.206,Z 172.957,A -85,B 0,C 180,E1 -2657.083,E2 -2657.083} C_VEL
LIN {X 0,Y 566.213,Z 172.954,A -85,B 0,C 180,E1 -2660.315,E2 -2660.315} C_VEL
LIN {X 0,Y 566.181,Z 172.958,A -85,B 0,C 180,E1 -2663.428,E2 -2663.428} C_VEL
LIN {X 0,Y 566.128,Z 172.982,A -85,B 0,C 180,E1 -2666.077,E2 -2666.077} C_VEL
LIN {X 0,Y 566.136,Z 182.116,A -85,B 0,C 180,E1 -2668.575,E2 -2668.575} C_VEL
LIN {X 0,Y 566.148,Z 191.961,A -85,B 0,C 180,E1 -2671.45,E2 -2671.45} C_VEL
LIN {X 0,Y 566.23,Z 201.007,A -85,B 0,C 180,E1 -2674.252,E2 -2674.252} C_VEL
LIN {X 0,Y 566.194,Z 208.561,A -85,B 0,C 180,E1 -2676.715,E2 -2676.715} C_VEL
LIN {X 0,Y 566.152,Z 216.4,A -85,B 0,C 180,E1 -2679.281,E2 -2679.281} C_VEL
LIN {X 0,Y 566.074,Z 224.01,A -85,B 0,C 180,E1 -2681.918,E2 -2681.918} C_VEL
LIN {X 0,Y 566.027,Z 231.799,A -85,B 0,C 180,E1 -2684.517,E2 -2684.517} C_VEL
LIN {X 0,Y 566.004,Z 240.493,A -85,B 0,C 180,E1 -2687.381,E2 -2687.381} C_VEL
LIN {X 0,Y 566.926,Z 247.479,A -85,B 0,C 180,E1 -2687.539,E2 -2687.539} C_VEL
LIN {X 0,Y 566.833,Z 259.88,A -85,B 0,C 180,E1 -2687.877,E2 -2687.877} C_VEL
LIN {X 0,Y 566.698,Z 271.846,A -85,B 0,C 180,E1 -2688.342,E2 -2688.342} C_VEL
LIN {X 0,Y 566.574,Z 283.595,A -85,B 0,C 180,E1 -2688.949,E2 -2688.949} C_VEL
LIN {X 0,Y 566.452,Z 294.117,A -85,B 0,C 180,E1 -2689.636,E2 -2689.636} C_VEL
LIN {X 0,Y 566.302,Z 303.134,A -85,B 0,C 180,E1 -2690.355,E2 -2690.355} C_VEL
LIN {X 0,Y 566.183,Z 312.375,A -85,B 0,C 180,E1 -2691.254,E2 -2691.254} C_VEL
LIN {X 0,Y 566.081,Z 321.36,A -85,B 0,C 180,E1 -2692.33,E2 -2692.33} C_VEL
LIN {X 0,Y 566.01,Z 328.459,A -85,B 0,C 180,E1 -2693.386,E2 -2693.386} C_VEL
LIN {X 0,Y 565.937,Z 335.18,A -85,B 0,C 180,E1 -2694.656,E2 -2694.656} C_VEL
LIN {X 0,Y 565.96,Z 339.536,A -85,B 0,C 180,E1 -2695.727,E2 -2695.727} C_VEL
LIN {X 0,Y 565.927,Z 341.834,A -85,B 0,C 180,E1 -2696.44,E2 -2696.44} C_VEL
LIN {X 0,Y 565.878,Z 343.69,A -85,B 0,C 180,E1 -2697.152,E2 -2697.152} C_VEL
LIN {X 0,Y 565.839,Z 345.135,A -85,B 0,C 180,E1 -2697.865,E2 -2697.865} C_VEL
LIN {X 0,Y 565.842,Z 346.755,A -85,B 0,C 180,E1 -2699.288,E2 -2699.288} C_VEL
LIN {X 0,Y 565.839,Z 346.996,A -85,B 0,C 180,E1 -2700,E2 -2700} C_VEL
LIN {X 0,Y 565.841,Z 346.813,A -85,B 0,C 180,E1 -2700.712,E2 -2700.712} C_VEL
LIN {X 0,Y 565.838,Z 345.274,A -85,B 0,C 180,E1 -2702.135,E2 -2702.135} C_VEL
LIN {X 0,Y 565.879,Z 343.906,A -85,B 0,C 180,E1 -2702.848,E2 -2702.848} C_VEL
LIN {X 0,Y 565.926,Z 341.037,A -85,B 0,C 180,E1 -2703.917,E2 -2703.917} C_VEL
LIN {X 0,Y 565.878,Z 337.136,A -85,B 0,C 180,E1 -2704.988,E2 -2704.988} C_VEL
LIN {X 0,Y 565.992,Z 332.091,A -85,B 0,C 180,E1 -2706.059,E2 -2706.059} C_VEL
LIN {X 0,Y 566.032,Z 325.756,A -85,B 0,C 180,E1 -2707.132,E2 -2707.132} C_VEL
LIN {X 0,Y 566.129,Z 317.865,A -85,B 0,C 180,E1 -2708.208,E2 -2708.208} C_VEL
LIN {X 0,Y 566.229,Z 309.788,A -85,B 0,C 180,E1 -2709.106,E2 -2709.106} C_VEL
LIN {X 0,Y 566.325,Z 299.926,A -85,B 0,C 180,E1 -2710.005,E2 -2710.005} C_VEL
LIN {X 0,Y 566.47,Z 289.028,A -85,B 0,C 180,E1 -2710.806,E2 -2710.806} C_VEL
LIN {X 0,Y 566.608,Z 276.851,A -85,B 0,C 180,E1 -2711.509,E2 -2711.509} C_VEL
LIN {X 0,Y 566.758,Z 264.965,A -85,B 0,C 180,E1 -2712.033,E2 -2712.033} C_VEL
LIN {X 0,Y 566.909,Z 251.312,A -85,B 0,C 180,E1 -2712.462,E2 -2712.462} C_VEL
LIN {X 0,Y 566.701,Z 245.158,A -85,B 0,C 180,E1 -2712.606,E2 -2712.606} C_VEL
LIN {X 0,Y 565.975,Z 240.49,A -85,B 0,C 180,E1 -2712.71,E2 -2712.71} C_VEL
LIN {X 0,Y 566.009,Z 230.957,A -85,B 0,C 180,E1 -2715.853,E2 -2715.853} C_VEL
LIN {X 0,Y 566.085,Z 221.911,A -85,B 0,C 180,E1 -2718.884,E2 -2718.884} C_VEL
LIN {X 0,Y 566.145,Z 213.329,A -85,B 0,C 180,E1 -2721.857,E2 -2721.857} C_VEL
LIN {X 0,Y 565.472,Z 211.72,A -85,B 0,C 180,E1 -2722.429,E2 -2722.429} C_VEL
LIN {X 0,Y 562.617,Z 209.291,A -85,B 0,C 180,E1 -2723.362,E2 -2723.362} C_VEL
LIN {X 0,Y 560.227,Z 207.37,A -85,B 0,C 180,E1 -2724.113,E2 -2724.113} C_VEL
LIN {X 0,Y 559.226,Z 205.818,A -85,B 0,C 180,E1 -2724.691,E2 -2724.691} C_VEL
LIN {X 0,Y 559.158,Z 205.268,A -85,B 0,C 180,E1 -2724.886,E2 -2724.886} C_VEL
LIN {X 0,Y 559.237,Z 196.927,A -85,B 0,C 180,E1 -2727.709,E2 -2727.709} C_VEL
LIN {X 0,Y 559.295,Z 188.501,A -85,B 0,C 180,E1 -2730.592,E2 -2730.592} C_VEL
LIN {X 0,Y 559.341,Z 181.076,A -85,B 0,C 180,E1 -2733.132,E2 -2733.132} C_VEL
LIN {X 0,Y 559.28,Z 174.671,A -85,B 0,C 180,E1 -2735.313,E2 -2735.313} C_VEL
LIN {X 0,Y 559.127,Z 173.841,A -85,B 0,C 180,E1 -2735.656,E2 -2735.656} C_VEL
LIN {X 0,Y 559.177,Z 173.83,A -85,B 0,C 180,E1 -2738.808,E2 -2738.808} C_VEL
LIN {X 0,Y 559.166,Z 173.831,A -85,B 0,C 180,E1 -2741.77,E2 -2741.77} C_VEL
LIN {X 0,Y 559.131,Z 173.836,A -85,B 0,C 180,E1 -2744.74,E2 -2744.74} C_VEL
LIN {X 0,Y 559.162,Z 173.835,A -85,B 0,C 180,E1 -2747.256,E2 -2747.256} C_VEL
LIN {X 0,Y 559.184,Z 173.829,A -85,B 0,C 180,E1 -2750.134,E2 -2750.134} C_VEL
LIN {X 0,Y 559.119,Z 173.838,A -85,B 0,C 180,E1 -2752.889,E2 -2752.889} C_VEL
LIN {X 0,Y 559.158,Z 173.833,A -85,B 0,C 180,E1 -2756.053,E2 -2756.053} C_VEL
LIN {X 0,Y 559.16,Z 173.836,A -85,B 0,C 180,E1 -2758.98,E2 -2758.98} C_VEL
LIN {X 0,Y 559.037,Z 173.853,A -85,B 0,C 180,E1 -2760.639,E2 -2760.639} C_VEL
LIN {X 0,Y 559.071,Z 175.848,A -85,B 0,C 180,E1 -2762.281,E2 -2762.281} C_VEL
LIN {X 0,Y 559.023,Z 179.21,A -85,B 0,C 180,E1 -2764.848,E2 -2764.848} C_VEL
LIN {X 0,Y 558.921,Z 183.105,A -85,B 0,C 180,E1 -2767.837,E2 -2767.837} C_VEL
LIN {X 0,Y 558.888,Z 187.19,A -85,B 0,C 180,E1 -2770.916,E2 -2770.916} C_VEL
LIN {X 0,Y 558.82,Z 191.308,A -85,B 0,C 180,E1 -2773.937,E2 -2773.937} C_VEL
LIN {X 0,Y 558.839,Z 194.354,A -85,B 0,C 180,E1 -2776.175,E2 -2776.175} C_VEL
LIN {X 0,Y 558.806,Z 198.398,A -85,B 0,C 180,E1 -2779.125,E2 -2779.125} C_VEL
LIN {X 0,Y 558.719,Z 202.593,A -85,B 0,C 180,E1 -2782.046,E2 -2782.046} C_VEL
LIN {X 0,Y 558.762,Z 203.454,A -85,B 0,C 180,E1 -2782.615,E2 -2782.615} C_VEL
LIN {X 0,Y 559.153,Z 210.021,A -85,B 0,C 180,E1 -2782.869,E2 -2782.869} C_VEL
LIN {X 0,Y 559.07,Z 218.066,A -85,B 0,C 180,E1 -2783.267,E2 -2783.267} C_VEL
LIN {X 0,Y 559.018,Z 225.787,A -85,B 0,C 180,E1 -2783.774,E2 -2783.774} C_VEL
LIN {X 0,Y 558.929,Z 231.354,A -85,B 0,C 180,E1 -2784.226,E2 -2784.226} C_VEL
LIN {X 0,Y 558.931,Z 238.308,A -85,B 0,C 180,E1 -2784.95,E2 -2784.95} C_VEL
LIN {X 0,Y 558.907,Z 243.749,A -85,B 0,C 180,E1 -2785.672,E2 -2785.672} C_VEL
LIN {X 0,Y 558.88,Z 248.035,A -85,B 0,C 180,E1 -2786.394,E2 -2786.394} C_VEL
LIN {X 0,Y 558.816,Z 251.372,A -85,B 0,C 180,E1 -2787.116,E2 -2787.116} C_VEL
LIN {X 0,Y 558.763,Z 253.863,A -85,B 0,C 180,E1 -2787.837,E2 -2787.837} C_VEL
LIN {X 0,Y 558.747,Z 255.567,A -85,B 0,C 180,E1 -2788.558,E2 -2788.558} C_VEL
LIN {X 0,Y 558.742,Z 256.563,A -85,B 0,C 180,E1 -2789.278,E2 -2789.278} C_VEL
LIN {X 0,Y 558.74,Z 256.927,A -85,B 0,C 180,E1 -2789.999,E2 -2789.999} C_VEL
LIN {X 0,Y 558.741,Z 256.668,A -85,B 0,C 180,E1 -2790.72,E2 -2790.72} C_VEL
LIN {X 0,Y 558.748,Z 255.76,A -85,B 0,C 180,E1 -2791.441,E2 -2791.441} C_VEL
LIN {X 0,Y 558.762,Z 254.116,A -85,B 0,C 180,E1 -2792.162,E2 -2792.162} C_VEL
LIN {X 0,Y 558.859,Z 250.238,A -85,B 0,C 180,E1 -2793.243,E2 -2793.243} C_VEL
LIN {X 0,Y 558.875,Z 245.483,A -85,B 0,C 180,E1 -2794.146,E2 -2794.146} C_VEL
LIN {X 0,Y 558.951,Z 240.519,A -85,B 0,C 180,E1 -2794.868,E2 -2794.868} C_VEL
LIN {X 0,Y 558.889,Z 234.145,A -85,B 0,C 180,E1 -2795.592,E2 -2795.592} C_VEL
LIN {X 0,Y 559,Z 228.146,A -85,B 0,C 180,E1 -2796.134,E2 -2796.134} C_VEL
LIN {X 0,Y 559.013,Z 221.85,A -85,B 0,C 180,E1 -2796.596,E2 -2796.596} C_VEL
LIN {X 0,Y 559.13,Z 213.363,A -85,B 0,C 180,E1 -2797.07,E2 -2797.07} C_VEL
LIN {X 0,Y 559.048,Z 206.716,A -85,B 0,C 180,E1 -2797.357,E2 -2797.357} C_VEL
LIN {X 0,Y 558.733,Z 203.455,A -85,B 0,C 180,E1 -2797.475,E2 -2797.475} C_VEL
LIN {X 0,Y 558.759,Z 199.527,A -85,B 0,C 180,E1 -2800.141,E2 -2800.141} C_VEL
LIN {X 0,Y 558.792,Z 196.472,A -85,B 0,C 180,E1 -2802.345,E2 -2802.345} C_VEL
LIN {X 0,Y 558.836,Z 193.502,A -85,B 0,C 180,E1 -2804.567,E2 -2804.567} C_VEL
LIN {X 0,Y 558.851,Z 189.397,A -85,B 0,C 180,E1 -2807.566,E2 -2807.566} C_VEL
LIN {X 0,Y 558.876,Z 186.338,A -85,B 0,C 180,E1 -2809.847,E2 -2809.847} C_VEL
LIN {X 0,Y 558.908,Z 183.241,A -85,B 0,C 180,E1 -2812.161,E2 -2812.161} C_VEL
LIN {X 0,Y 559.016,Z 179.355,A -85,B 0,C 180,E1 -2815.15,E2 -2815.15} C_VEL
LIN {X 0,Y 559.056,Z 175.994,A -85,B 0,C 180,E1 -2817.718,E2 -2817.718} C_VEL
LIN {X 0,Y 559.03,Z 173.854,A -85,B 0,C 180,E1 -2819.359,E2 -2819.359} C_VEL
LIN {X 0,Y 559.16,Z 173.835,A -85,B 0,C 180,E1 -2821.862,E2 -2821.862} C_VEL
LIN {X 0,Y 559.143,Z 173.831,A -85,B 0,C 180,E1 -2824.444,E2 -2824.444} C_VEL
LIN {X 0,Y 559.139,Z 173.836,A -85,B 0,C 180,E1 -2827.107,E2 -2827.107} C_VEL
LIN {X 0,Y 559.159,Z 173.83,A -85,B 0,C 180,E1 -2829.941,E2 -2829.941} C_VEL
LIN {X 0,Y 559.154,Z 173.833,A -85,B 0,C 180,E1 -2832.742,E2 -2832.742} C_VEL
LIN {X 0,Y 559.147,Z 173.831,A -85,B 0,C 180,E1 -2835.76,E2 -2835.76} C_VEL
LIN {X 0,Y 559.185,Z 173.827,A -85,B 0,C 180,E1 -2838.232,E2 -2838.232} C_VEL
LIN {X 0,Y 559.171,Z 173.83,A -85,B 0,C 180,E1 -2841.19,E2 -2841.19} C_VEL
LIN {X 0,Y 559.165,Z 173.828,A -85,B 0,C 180,E1 -2843.791,E2 -2843.791} C_VEL
LIN {X 0,Y 559.17,Z 173.835,A -85,B 0,C 180,E1 -2846.425,E2 -2846.425} C_VEL
LIN {X 0,Y 559.158,Z 173.83,A -85,B 0,C 180,E1 -2848.981,E2 -2848.981} C_VEL
LIN {X 0,Y 559.162,Z 173.829,A -85,B 0,C 180,E1 -2851.617,E2 -2851.617} C_VEL
LIN {X 0,Y 559.19,Z 173.83,A -85,B 0,C 180,E1 -2853.903,E2 -2853.903} C_VEL
LIN {X 0,Y 559.148,Z 173.833,A -85,B 0,C 180,E1 -2856.566,E2 -2856.566} C_VEL
LIN {X 0,Y 559.177,Z 173.828,A -85,B 0,C 180,E1 -2859.395,E2 -2859.395} C_VEL
LIN {X 0,Y 559.145,Z 173.837,A -85,B 0,C 180,E1 -2861.686,E2 -2861.686} C_VEL
LIN {X 0,Y 559.162,Z 173.832,A -85,B 0,C 180,E1 -2863.948,E2 -2863.948} C_VEL
LIN {X 0,Y 559.164,Z 173.83,A -85,B 0,C 180,E1 -2866.184,E2 -2866.184} C_VEL
LIN {X 0,Y 559.199,Z 173.828,A -85,B 0,C 180,E1 -2869.134,E2 -2869.134} C_VEL
LIN {X 0,Y 559.199,Z 173.824,A -85,B 0,C 180,E1 -2872.053,E2 -2872.053} C_VEL
LIN {X 0,Y 559.246,Z 173.822,A -85,B 0,C 180,E1 -2874.953,E2 -2874.953} C_VEL
LIN {X 0,Y 559.232,Z 173.82,A -85,B 0,C 180,E1 -2877.839,E2 -2877.839} C_VEL
LIN {X 0,Y 559.268,Z 173.819,A -85,B 0,C 180,E1 -2880.72,E2 -2880.72} C_VEL
LIN {X 0,Y 559.23,Z 173.828,A -85,B 0,C 180,E1 -2882.881,E2 -2882.881} C_VEL
LIN {X 0,Y 559.205,Z 173.823,A -85,B 0,C 180,E1 -2885.77,E2 -2885.77} C_VEL
LIN {X 0,Y 559.176,Z 173.833,A -85,B 0,C 180,E1 -2888.675,E2 -2888.675} C_VEL
LIN {X 0,Y 559.191,Z 173.825,A -85,B 0,C 180,E1 -2891.601,E2 -2891.601} C_VEL
LIN {X 0,Y 559.188,Z 173.83,A -85,B 0,C 180,E1 -2894.596,E2 -2894.596} C_VEL
LIN {X 0,Y 559.119,Z 173.834,A -85,B 0,C 180,E1 -2897.558,E2 -2897.558} C_VEL
LIN {X 0,Y 559.15,Z 173.836,A -85,B 0,C 180,E1 -2899.838,E2 -2899.838} C_VEL
LIN {X 0,Y 559.117,Z 173.841,A -85,B 0,C 180,E1 -2902.154,E2 -2902.154} C_VEL
LIN {X 0,Y 559.126,Z 173.835,A -85,B 0,C 180,E1 -2905.178,E2 -2905.178} C_VEL
LIN {X 0,Y 559.088,Z 173.847,A -85,B 0,C 180,E1 -2907.717,E2 -2907.717} C_VEL
LIN {X 0,Y 559.119,Z 173.836,A -85,B 0,C 180,E1 -2910.185,E2 -2910.185} C_VEL
LIN {X 0,Y 559.139,Z 173.832,A -85,B 0,C 180,E1 -2912.716,E2 -2912.716} C_VEL
LIN {X 0,Y 559.107,Z 173.844,A -85,B 0,C 180,E1 -2915.326,E2 -2915.326} C_VEL
LIN {X 0,Y 559.117,Z 173.836,A -85,B 0,C 180,E1 -2918.019,E2 -2918.019} C_VEL
LIN {X 0,Y 559.144,Z 173.835,A -85,B 0,C 180,E1 -2920.814,E2 -2920.814} C_VEL
LIN {X 0,Y 559.128,Z 173.834,A -85,B 0,C 180,E1 -2923.735,E2 -2923.735} C_VEL
LIN {X 0,Y 559.138,Z 173.84,A -85,B 0,C 180,E1 -2926.805,E2 -2926.805} C_VEL
LIN {X 0,Y 559.148,Z 173.834,A -85,B 0,C 180,E1 -2929.189,E2 -2929.189} C_VEL
LIN {X 0,Y 559.126,Z 173.836,A -85,B 0,C 180,E1 -2931.983,E2 -2931.983} C_VEL
LIN {X 0,Y 559.129,Z 173.837,A -85,B 0,C 180,E1 -2934.788,E2 -2934.788} C_VEL
LIN {X 0,Y 559.152,Z 173.833,A -85,B 0,C 180,E1 -2937.365,E2 -2937.365} C_VEL
LIN {X 0,Y 559.135,Z 173.842,A -85,B 0,C 180,E1 -2939.4,E2 -2939.4} C_VEL
LIN {X 0,Y 561.038,Z 182.681,A -85,B 0,C 180,E1 -2940.933,E2 -2940.933} C_VEL
LIN {X 0,Y 560.643,Z 198.523,A -85,B 0,C 180,E1 -2943.376,E2 -2943.376} C_VEL
LIN {X 0,Y 560.299,Z 217.361,A -85,B 0,C 180,E1 -2946.16,E2 -2946.16} C_VEL
LIN {X 0,Y 560.014,Z 236.044,A -85,B 0,C 180,E1 -2948.852,E2 -2948.852} C_VEL
LIN {X 0,Y 559.777,Z 257.853,A -85,B 0,C 180,E1 -2951.898,E2 -2951.898} C_VEL
LIN {X 0,Y 559.452,Z 277.797,A -85,B 0,C 180,E1 -2954.705,E2 -2954.705} C_VEL
LIN {X 0,Y 559.302,Z 294.915,A -85,B 0,C 180,E1 -2957.09,E2 -2957.09} C_VEL
LIN {X 0,Y 560.075,Z 301.678,A -85,B 0,C 180,E1 -2957.224,E2 -2957.224} C_VEL
LIN {X 0,Y 559.925,Z 314.722,A -85,B 0,C 180,E1 -2957.52,E2 -2957.52} C_VEL
LIN {X 0,Y 559.805,Z 327.268,A -85,B 0,C 180,E1 -2957.954,E2 -2957.954} C_VEL
LIN {X 0,Y 559.667,Z 339.831,A -85,B 0,C 180,E1 -2958.548,E2 -2958.548} C_VEL
LIN {X 0,Y 559.49,Z 350.922,A -85,B 0,C 180,E1 -2959.232,E2 -2959.232} C_VEL
LIN {X 0,Y 559.315,Z 361.55,A -85,B 0,C 180,E1 -2960.052,E2 -2960.052} C_VEL
LIN {X 0,Y 559.161,Z 371.123,A -85,B 0,C 180,E1 -2960.962,E2 -2960.962} C_VEL
LIN {X 0,Y 559.049,Z 378.968,A -85,B 0,C 180,E1 -2961.871,E2 -2961.871} C_VEL
LIN {X 0,Y 558.942,Z 386.629,A -85,B 0,C 180,E1 -2962.959,E2 -2962.959} C_VEL
LIN {X 0,Y 558.935,Z 393.684,A -85,B 0,C 180,E1 -2964.228,E2 -2964.228} C_VEL
LIN {X 0,Y 558.826,Z 398.376,A -85,B 0,C 180,E1 -2965.312,E2 -2965.312} C_VEL
LIN {X 0,Y 558.836,Z 401.963,A -85,B 0,C 180,E1 -2966.396,E2 -2966.396} C_VEL
LIN {X 0,Y 558.799,Z 403.812,A -85,B 0,C 180,E1 -2967.117,E2 -2967.117} C_VEL
LIN {X 0,Y 558.745,Z 406.186,A -85,B 0,C 180,E1 -2968.559,E2 -2968.559} C_VEL
LIN {X 0,Y 558.74,Z 407,A -85,B 0,C 180,E1 -2970.001,E2 -2970.001} C_VEL
LIN {X 0,Y 558.745,Z 406.183,A -85,B 0,C 180,E1 -2971.442,E2 -2971.442} C_VEL
LIN {X 0,Y 558.799,Z 403.806,A -85,B 0,C 180,E1 -2972.885,E2 -2972.885} C_VEL
LIN {X 0,Y 558.844,Z 400.892,A -85,B 0,C 180,E1 -2973.967,E2 -2973.967} C_VEL
LIN {X 0,Y 558.798,Z 396.946,A -85,B 0,C 180,E1 -2975.052,E2 -2975.052} C_VEL
LIN {X 0,Y 558.922,Z 391.863,A -85,B 0,C 180,E1 -2976.136,E2 -2976.136} C_VEL
LIN {X 0,Y 558.978,Z 385.461,A -85,B 0,C 180,E1 -2977.224,E2 -2977.224} C_VEL
LIN {X 0,Y 559.097,Z 377.471,A -85,B 0,C 180,E1 -2978.313,E2 -2978.313} C_VEL
LIN {X 0,Y 559.195,Z 369.326,A -85,B 0,C 180,E1 -2979.222,E2 -2979.222} C_VEL
LIN {X 0,Y 559.357,Z 359.39,A -85,B 0,C 180,E1 -2980.132,E2 -2980.132} C_VEL
LIN {X 0,Y 559.552,Z 348.391,A -85,B 0,C 180,E1 -2980.937,E2 -2980.937} C_VEL
LIN {X 0,Y 559.673,Z 336.444,A -85,B 0,C 180,E1 -2981.629,E2 -2981.629} C_VEL
LIN {X 0,Y 559.828,Z 323.753,A -85,B 0,C 180,E1 -2982.185,E2 -2982.185} C_VEL
LIN {X 0,Y 559.965,Z 310.319,A -85,B 0,C 180,E1 -2982.597,E2 -2982.597} C_VEL
LIN {X 0,Y 559.981,Z 300.054,A -85,B 0,C 180,E1 -2982.803,E2 -2982.803} C_VEL
LIN {X 0,Y 559.304,Z 294.902,A -85,B 0,C 180,E1 -2982.912,E2 -2982.912} C_VEL
LIN {X 0,Y 559.511,Z 275.124,A -85,B 0,C 180,E1 -2985.669,E2 -2985.669} C_VEL
LIN {X 0,Y 559.756,Z 255.155,A -85,B 0,C 180,E1 -2988.484,E2 -2988.484} C_VEL
LIN {X 0,Y 559.963,Z 237.449,A -85,B 0,C 180,E1 -2990.96,E2 -2990.96} C_VEL
LIN {X 0,Y 560.247,Z 219.9,A -85,B 0,C 180,E1 -2993.472,E2 -2993.472} C_VEL
LIN {X 0,Y 560.628,Z 199.823,A -85,B 0,C 180,E1 -2996.426,E2 -2996.426} C_VEL
LIN {X 0,Y 561.039,Z 183.545,A -85,B 0,C 180,E1 -2998.924,E2 -2998.924} C_VEL
LIN {X 0,Y 560.343,Z 179.079,A -85,B 0,C 180,E1 -2999.667,E2 -2999.667} C_VEL
LIN {X 0,Y 559.136,Z 173.839,A -85,B 0,C 180,E1 -3000.602,E2 -3000.602} C_VEL
LIN {X 0,Y 559.139,Z 173.839,A -85,B 0,C 180,E1 -3002.717,E2 -3002.717} C_VEL
LIN {X 0,Y 559.119,Z 173.841,A -85,B 0,C 180,E1 -3005.325,E2 -3005.325} C_VEL
LIN {X 0,Y 559.132,Z 173.837,A -85,B 0,C 180,E1 -3008.018,E2 -3008.018} C_VEL
LIN {X 0,Y 559.16,Z 173.832,A -85,B 0,C 180,E1 -3010.813,E2 -3010.813} C_VEL
LIN {X 0,Y 559.143,Z 173.84,A -85,B 0,C 180,E1 -3013.734,E2 -3013.734} C_VEL
LIN {X 0,Y 559.15,Z 173.833,A -85,B 0,C 180,E1 -3016.804,E2 -3016.804} C_VEL
LIN {X 0,Y 559.16,Z 173.838,A -85,B 0,C 180,E1 -3019.188,E2 -3019.188} C_VEL
LIN {X 0,Y 559.13,Z 173.836,A -85,B 0,C 180,E1 -3021.982,E2 -3021.982} C_VEL
LIN {X 0,Y 559.117,Z 173.843,A -85,B 0,C 180,E1 -3024.79,E2 -3024.79} C_VEL
LIN {X 0,Y 559.087,Z 173.883,A -85,B 0,C 180,E1 -3026.064,E2 -3026.064} C_VEL
LIN {X 0,Y 559.08,Z 183.613,A -85,B 0,C 180,E1 -3028.739,E2 -3028.739} C_VEL
LIN {X 0,Y 559.11,Z 193.447,A -85,B 0,C 180,E1 -3031.631,E2 -3031.631} C_VEL
LIN {X 0,Y 559.177,Z 202.034,A -85,B 0,C 180,E1 -3034.303,E2 -3034.303} C_VEL
LIN {X 0,Y 559.13,Z 210.54,A -85,B 0,C 180,E1 -3037.067,E2 -3037.067} C_VEL
LIN {X 0,Y 559.115,Z 218.751,A -85,B 0,C 180,E1 -3039.777,E2 -3039.777} C_VEL
LIN {X 0,Y 559.005,Z 227.497,A -85,B 0,C 180,E1 -3042.844,E2 -3042.844} C_VEL
LIN {X 0,Y 558.946,Z 236.342,A -85,B 0,C 180,E1 -3045.837,E2 -3045.837} C_VEL
LIN {X 0,Y 558.935,Z 240.7,A -85,B 0,C 180,E1 -3047.231,E2 -3047.231} C_VEL
LIN {X 0,Y 559.985,Z 248.496,A -85,B 0,C 180,E1 -3047.405,E2 -3047.405} C_VEL
LIN {X 0,Y 559.895,Z 261.261,A -85,B 0,C 180,E1 -3047.771,E2 -3047.771} C_VEL
LIN {X 0,Y 559.71,Z 272.928,A -85,B 0,C 180,E1 -3048.245,E2 -3048.245} C_VEL
LIN {X 0,Y 559.565,Z 285.308,A -85,B 0,C 180,E1 -3048.91,E2 -3048.91} C_VEL
LIN {X 0,Y 559.401,Z 296.52,A -85,B 0,C 180,E1 -3049.687,E2 -3049.687} C_VEL
LIN {X 0,Y 559.239,Z 307.071,A -85,B 0,C 180,E1 -3050.597,E2 -3050.597} C_VEL
LIN {X 0,Y 559.129,Z 315.606,A -85,B 0,C 180,E1 -3051.507,E2 -3051.507} C_VEL
LIN {X 0,Y 558.975,Z 323.936,A -85,B 0,C 180,E1 -3052.596,E2 -3052.596} C_VEL
LIN {X 0,Y 558.895,Z 329.616,A -85,B 0,C 180,E1 -3053.502,E2 -3053.502} C_VEL
LIN {X 0,Y 558.869,Z 335.184,A -85,B 0,C 180,E1 -3054.588,E2 -3054.588} C_VEL
LIN {X 0,Y 558.869,Z 339.541,A -85,B 0,C 180,E1 -3055.673,E2 -3055.673} C_VEL
LIN {X 0,Y 558.836,Z 341.834,A -85,B 0,C 180,E1 -3056.395,E2 -3056.395} C_VEL
LIN {X 0,Y 558.799,Z 343.689,A -85,B 0,C 180,E1 -3057.116,E2 -3057.116} C_VEL
LIN {X 0,Y 558.745,Z 345.136,A -85,B 0,C 180,E1 -3057.837,E2 -3057.837} C_VEL
LIN {X 0,Y 558.742,Z 346.755,A -85,B 0,C 180,E1 -3059.279,E2 -3059.279} C_VEL
LIN {X 0,Y 558.74,Z 346.996,A -85,B 0,C 180,E1 -3060,E2 -3060} C_VEL
LIN {X 0,Y 558.741,Z 346.812,A -85,B 0,C 180,E1 -3060.721,E2 -3060.721} C_VEL
LIN {X 0,Y 558.745,Z 345.274,A -85,B 0,C 180,E1 -3062.163,E2 -3062.163} C_VEL
LIN {X 0,Y 558.8,Z 343.903,A -85,B 0,C 180,E1 -3062.884,E2 -3062.884} C_VEL
LIN {X 0,Y 558.844,Z 341.034,A -85,B 0,C 180,E1 -3063.966,E2 -3063.966} C_VEL
LIN {X 0,Y 558.798,Z 337.131,A -85,B 0,C 180,E1 -3065.051,E2 -3065.051} C_VEL
LIN {X 0,Y 558.912,Z 332.086,A -85,B 0,C 180,E1 -3066.136,E2 -3066.136} C_VEL
LIN {X 0,Y 558.973,Z 325.75,A -85,B 0,C 180,E1 -3067.223,E2 -3067.223} C_VEL
LIN {X 0,Y 559.091,Z 317.863,A -85,B 0,C 180,E1 -3068.312,E2 -3068.312} C_VEL
LIN {X 0,Y 559.182,Z 309.78,A -85,B 0,C 180,E1 -3069.221,E2 -3069.221} C_VEL
LIN {X 0,Y 559.335,Z 299.917,A -85,B 0,C 180,E1 -3070.132,E2 -3070.132} C_VEL
LIN {X 0,Y 559.481,Z 289.121,A -85,B 0,C 180,E1 -3070.936,E2 -3070.936} C_VEL
LIN {X 0,Y 559.653,Z 276.47,A -85,B 0,C 180,E1 -3071.674,E2 -3071.674} C_VEL
LIN {X 0,Y 559.827,Z 264.942,A -85,B 0,C 180,E1 -3072.185,E2 -3072.185} C_VEL
LIN {X 0,Y 559.981,Z 251.282,A -85,B 0,C 180,E1 -3072.618,E2 -3072.618} C_VEL
LIN {X 0,Y 559.7,Z 245.703,A -85,B 0,C 180,E1 -3072.755,E2 -3072.755} C_VEL
LIN {X 0,Y 558.913,Z 240.488,A -85,B 0,C 180,E1 -3072.874,E2 -3072.874} C_VEL
LIN {X 0,Y 558.937,Z 230.955,A -85,B 0,C 180,E1 -3076.059,E2 -3076.059} C_VEL
LIN {X 0,Y 559.055,Z 222.2,A -85,B 0,C 180,E1 -3079.078,E2 -3079.078} C_VEL
LIN {X 0,Y 559.112,Z 214.105,A -85,B 0,C 180,E1 -3081.883,E2 -3081.883} C_VEL
LIN {X 0,Y 559.143,Z 206.359,A -85,B 0,C 180,E1 -3084.506,E2 -3084.506} C_VEL
LIN {X 0,Y 559.158,Z 205.268,A -85,B 0,C 180,E1 -3084.886,E2 -3084.886} C_VEL
LIN {X 0,Y 558.531,Z 203.691,A -85,B 0,C 180,E1 -3085.465,E2 -3085.465} C_VEL
LIN {X 0,Y 555.708,Z 201.237,A -85,B 0,C 180,E1 -3086.41,E2 -3086.41} C_VEL
LIN {X 0,Y 553.3,Z 199.292,A -85,B 0,C 180,E1 -3087.17,E2 -3087.17} C_VEL
LIN {X 0,Y 552.261,Z 197.705,A -85,B 0,C 180,E1 -3087.754,E2 -3087.754} C_VEL
LIN {X 0,Y 552.174,Z 197.139,A -85,B 0,C 180,E1 -3087.951,E2 -3087.951} C_VEL
LIN {X 0,Y 552.289,Z 188.285,A -85,B 0,C 180,E1 -3091.022,E2 -3091.022} C_VEL
LIN {X 0,Y 552.307,Z 180.832,A -85,B 0,C 180,E1 -3093.61,E2 -3093.61} C_VEL
LIN {X 0,Y 552.217,Z 175.407,A -85,B 0,C 180,E1 -3095.459,E2 -3095.459} C_VEL
LIN {X 0,Y 552.103,Z 174.716,A -85,B 0,C 180,E1 -3095.73,E2 -3095.73} C_VEL
LIN {X 0,Y 552.119,Z 174.709,A -85,B 0,C 180,E1 -3098.589,E2 -3098.589} C_VEL
LIN {X 0,Y 552.125,Z 174.71,A -85,B 0,C 180,E1 -3101.446,E2 -3101.446} C_VEL
LIN {X 0,Y 552.08,Z 174.716,A -85,B 0,C 180,E1 -3104.529,E2 -3104.529} C_VEL
LIN {X 0,Y 552.135,Z 174.712,A -85,B 0,C 180,E1 -3107.584,E2 -3107.584} C_VEL
LIN {X 0,Y 552.134,Z 174.71,A -85,B 0,C 180,E1 -3110.472,E2 -3110.472} C_VEL
LIN {X 0,Y 552.073,Z 174.716,A -85,B 0,C 180,E1 -3113.322,E2 -3113.322} C_VEL
LIN {X 0,Y 552.103,Z 174.713,A -85,B 0,C 180,E1 -3115.937,E2 -3115.937} C_VEL
LIN {X 0,Y 552.126,Z 174.712,A -85,B 0,C 180,E1 -3118.54,E2 -3118.54} C_VEL
LIN {X 0,Y 552.049,Z 174.723,A -85,B 0,C 180,E1 -3120.231,E2 -3120.231} C_VEL
LIN {X 0,Y 551.968,Z 174.972,A -85,B 0,C 180,E1 -3121.063,E2 -3121.063} C_VEL
LIN {X 0,Y 551.975,Z 178.321,A -85,B 0,C 180,E1 -3123.535,E2 -3123.535} C_VEL
LIN {X 0,Y 551.919,Z 181.401,A -85,B 0,C 180,E1 -3125.953,E2 -3125.953} C_VEL
LIN {X 0,Y 551.875,Z 184.544,A -85,B 0,C 180,E1 -3128.379,E2 -3128.379} C_VEL
LIN {X 0,Y 551.8,Z 188.6,A -85,B 0,C 180,E1 -3131.432,E2 -3131.432} C_VEL
LIN {X 0,Y 551.755,Z 191.711,A -85,B 0,C 180,E1 -3133.726,E2 -3133.726} C_VEL
LIN {X 0,Y 551.783,Z 194.84,A -85,B 0,C 180,E1 -3135.995,E2 -3135.995} C_VEL
LIN {X 0,Y 551.76,Z 198.915,A -85,B 0,C 180,E1 -3138.984,E2 -3138.984} C_VEL
LIN {X 0,Y 551.704,Z 203.843,A -85,B 0,C 180,E1 -3142.496,E2 -3142.496} C_VEL
LIN {X 0,Y 552.148,Z 211.065,A -85,B 0,C 180,E1 -3142.778,E2 -3142.778} C_VEL
LIN {X 0,Y 552.064,Z 219.294,A -85,B 0,C 180,E1 -3143.205,E2 -3143.205} C_VEL
LIN {X 0,Y 552.003,Z 226.665,A -85,B 0,C 180,E1 -3143.708,E2 -3143.708} C_VEL
LIN {X 0,Y 551.891,Z 231.95,A -85,B 0,C 180,E1 -3144.152,E2 -3144.152} C_VEL
LIN {X 0,Y 551.889,Z 238.754,A -85,B 0,C 180,E1 -3144.885,E2 -3144.885} C_VEL
LIN {X 0,Y 551.848,Z 244.081,A -85,B 0,C 180,E1 -3145.617,E2 -3145.617} C_VEL
LIN {X 0,Y 551.794,Z 248.27,A -85,B 0,C 180,E1 -3146.348,E2 -3146.348} C_VEL
LIN {X 0,Y 551.742,Z 251.539,A -85,B 0,C 180,E1 -3147.079,E2 -3147.079} C_VEL
LIN {X 0,Y 551.675,Z 253.984,A -85,B 0,C 180,E1 -3147.809,E2 -3147.809} C_VEL
LIN {X 0,Y 551.649,Z 255.662,A -85,B 0,C 180,E1 -3148.539,E2 -3148.539} C_VEL
LIN {X 0,Y 551.643,Z 256.63,A -85,B 0,C 180,E1 -3149.269,E2 -3149.269} C_VEL
LIN {X 0,Y 551.641,Z 256.982,A -85,B 0,C 180,E1 -3149.999,E2 -3149.999} C_VEL
LIN {X 0,Y 551.642,Z 256.731,A -85,B 0,C 180,E1 -3150.729,E2 -3150.729} C_VEL
LIN {X 0,Y 551.649,Z 255.841,A -85,B 0,C 180,E1 -3151.459,E2 -3151.459} C_VEL
LIN {X 0,Y 551.674,Z 254.228,A -85,B 0,C 180,E1 -3152.189,E2 -3152.189} C_VEL
LIN {X 0,Y 551.785,Z 250.423,A -85,B 0,C 180,E1 -3153.285,E2 -3153.285} C_VEL
LIN {X 0,Y 551.805,Z 245.781,A -85,B 0,C 180,E1 -3154.199,E2 -3154.199} C_VEL
LIN {X 0,Y 551.897,Z 240.91,A -85,B 0,C 180,E1 -3154.93,E2 -3154.93} C_VEL
LIN {X 0,Y 551.86,Z 234.691,A -85,B 0,C 180,E1 -3155.663,E2 -3155.663} C_VEL
LIN {X 0,Y 551.984,Z 229.139,A -85,B 0,C 180,E1 -3156.185,E2 -3156.185} C_VEL
LIN {X 0,Y 552.026,Z 221.341,A -85,B 0,C 180,E1 -3156.762,E2 -3156.762} C_VEL
LIN {X 0,Y 552.147,Z 213.053,A -85,B 0,C 180,E1 -3157.22,E2 -3157.22} C_VEL
LIN {X 0,Y 551.986,Z 206.574,A -85,B 0,C 180,E1 -3157.498,E2 -3157.498} C_VEL
LIN {X 0,Y 551.662,Z 203.799,A -85,B 0,C 180,E1 -3157.617,E2 -3157.617} C_VEL
LIN {X 0,Y 551.756,Z 199.069,A -85,B 0,C 180,E1 -3161.014,E2 -3161.014} C_VEL
LIN {X 0,Y 551.768,Z 194.96,A -85,B 0,C 180,E1 -3164.004,E2 -3164.004} C_VEL
LIN {X 0,Y 551.784,Z 190.594,A -85,B 0,C 180,E1 -3167.202,E2 -3167.202} C_VEL
LIN {X 0,Y 551.831,Z 186.68,A -85,B 0,C 180,E1 -3170.111,E2 -3170.111} C_VEL
LIN {X 0,Y 551.861,Z 183.596,A -85,B 0,C 180,E1 -3172.46,E2 -3172.46} C_VEL
LIN {X 0,Y 551.972,Z 179.936,A -85,B 0,C 180,E1 -3175.309,E2 -3175.309} C_VEL
LIN {X 0,Y 551.991,Z 176.243,A -85,B 0,C 180,E1 -3178.104,E2 -3178.104} C_VEL
LIN {X 0,Y 551.992,Z 175.114,A -85,B 0,C 180,E1 -3178.934,E2 -3178.934} C_VEL
LIN {X 0,Y 552.058,Z 174.719,A -85,B 0,C 180,E1 -3180.039,E2 -3180.039} C_VEL
LIN {X 0,Y 552.113,Z 174.708,A -85,B 0,C 180,E1 -3182.845,E2 -3182.845} C_VEL
LIN {X 0,Y 552.088,Z 174.719,A -85,B 0,C 180,E1 -3185.441,E2 -3185.441} C_VEL
LIN {X 0,Y 552.091,Z 174.712,A -85,B 0,C 180,E1 -3187.885,E2 -3187.885} C_VEL
LIN {X 0,Y 552.113,Z 174.707,A -85,B 0,C 180,E1 -3190.479,E2 -3190.479} C_VEL
LIN {X 0,Y 552.108,Z 174.711,A -85,B 0,C 180,E1 -3193.483,E2 -3193.483} C_VEL
LIN {X 0,Y 552.104,Z 174.711,A -85,B 0,C 180,E1 -3196.576,E2 -3196.576} C_VEL
LIN {X 0,Y 552.115,Z 174.707,A -85,B 0,C 180,E1 -3199.519,E2 -3199.519} C_VEL
LIN {X 0,Y 552.086,Z 174.714,A -85,B 0,C 180,E1 -3202.335,E2 -3202.335} C_VEL
LIN {X 0,Y 552.123,Z 174.708,A -85,B 0,C 180,E1 -3205.054,E2 -3205.054} C_VEL
LIN {X 0,Y 552.12,Z 174.706,A -85,B 0,C 180,E1 -3207.681,E2 -3207.681} C_VEL
LIN {X 0,Y 552.137,Z 174.711,A -85,B 0,C 180,E1 -3210.236,E2 -3210.236} C_VEL
LIN {X 0,Y 552.138,Z 174.704,A -85,B 0,C 180,E1 -3212.997,E2 -3212.997} C_VEL
LIN {X 0,Y 552.104,Z 174.706,A -85,B 0,C 180,E1 -3215.161,E2 -3215.161} C_VEL
LIN {X 0,Y 552.087,Z 174.713,A -85,B 0,C 180,E1 -3217.549,E2 -3217.549} C_VEL
LIN {X 0,Y 552.139,Z 174.705,A -85,B 0,C 180,E1 -3220.372,E2 -3220.372} C_VEL
LIN {X 0,Y 552.148,Z 174.703,A -85,B 0,C 180,E1 -3222.977,E2 -3222.977} C_VEL
LIN {X 0,Y 552.127,Z 174.708,A -85,B 0,C 180,E1 -3226.004,E2 -3226.004} C_VEL
LIN {X 0,Y 552.167,Z 174.702,A -85,B 0,C 180,E1 -3228.993,E2 -3228.993} C_VEL
LIN {X 0,Y 552.153,Z 174.703,A -85,B 0,C 180,E1 -3231.951,E2 -3231.951} C_VEL
LIN {X 0,Y 552.22,Z 174.697,A -85,B 0,C 180,E1 -3234.889,E2 -3234.889} C_VEL
LIN {X 0,Y 552.205,Z 174.696,A -85,B 0,C 180,E1 -3237.812,E2 -3237.812} C_VEL
LIN {X 0,Y 552.237,Z 174.695,A -85,B 0,C 180,E1 -3240.729,E2 -3240.729} C_VEL
LIN {X 0,Y 552.195,Z 174.704,A -85,B 0,C 180,E1 -3242.918,E2 -3242.918} C_VEL
LIN {X 0,Y 552.176,Z 174.698,A -85,B 0,C 180,E1 -3245.844,E2 -3245.844} C_VEL
LIN {X 0,Y 552.142,Z 174.707,A -85,B 0,C 180,E1 -3248.786,E2 -3248.786} C_VEL
LIN {X 0,Y 552.148,Z 174.703,A -85,B 0,C 180,E1 -3251.751,E2 -3251.751} C_VEL
LIN {X 0,Y 552.123,Z 174.709,A -85,B 0,C 180,E1 -3254.749,E2 -3254.749} C_VEL
LIN {X 0,Y 552.078,Z 174.714,A -85,B 0,C 180,E1 -3257.79,E2 -3257.79} C_VEL
LIN {X 0,Y 552.111,Z 174.716,A -85,B 0,C 180,E1 -3260.102,E2 -3260.102} C_VEL
LIN {X 0,Y 552.069,Z 174.715,A -85,B 0,C 180,E1 -3262.452,E2 -3262.452} C_VEL
LIN {X 0,Y 552.069,Z 174.715,A -85,B 0,C 180,E1 -3265.335,E2 -3265.335} C_VEL
LIN {X 0,Y 552.036,Z 174.72,A -85,B 0,C 180,E1 -3268.102,E2 -3268.102} C_VEL
LIN {X 0,Y 552.078,Z 174.711,A -85,B 0,C 180,E1 -3270.611,E2 -3270.611} C_VEL
LIN {X 0,Y 552.101,Z 174.713,A -85,B 0,C 180,E1 -3273.187,E2 -3273.187} C_VEL
LIN {X 0,Y 552.06,Z 174.716,A -85,B 0,C 180,E1 -3275.846,E2 -3275.846} C_VEL
LIN {X 0,Y 552.103,Z 174.711,A -85,B 0,C 180,E1 -3278.59,E2 -3278.59} C_VEL
LIN {X 0,Y 552.1,Z 174.713,A -85,B 0,C 180,E1 -3281.448,E2 -3281.448} C_VEL
LIN {X 0,Y 552.08,Z 174.715,A -85,B 0,C 180,E1 -3284.532,E2 -3284.532} C_VEL
LIN {X 0,Y 552.123,Z 174.704,A -85,B 0,C 180,E1 -3287.586,E2 -3287.586} C_VEL
LIN {X 0,Y 552.126,Z 174.712,A -85,B 0,C 180,E1 -3290.474,E2 -3290.474} C_VEL
LIN {X 0,Y 552.101,Z 174.709,A -85,B 0,C 180,E1 -3293.318,E2 -3293.318} C_VEL
LIN {X 0,Y 552.123,Z 174.709,A -85,B 0,C 180,E1 -3295.94,E2 -3295.94} C_VEL
LIN {X 0,Y 552.128,Z 174.712,A -85,B 0,C 180,E1 -3299.075,E2 -3299.075} C_VEL
LIN {X 0,Y 552.146,Z 174.998,A -85,B 0,C 180,E1 -3299.183,E2 -3299.183} C_VEL
LIN {X 0,Y 554.126,Z 183.808,A -85,B 0,C 180,E1 -3300.761,E2 -3300.761} C_VEL
LIN {X 0,Y 553.803,Z 198.242,A -85,B 0,C 180,E1 -3303.021,E2 -3303.021} C_VEL
LIN {X 0,Y 553.386,Z 216.873,A -85,B 0,C 180,E1 -3305.823,E2 -3305.823} C_VEL
LIN {X 0,Y 553.104,Z 234.344,A -85,B 0,C 180,E1 -3308.379,E2 -3308.379} C_VEL
LIN {X 0,Y 552.798,Z 251.927,A -85,B 0,C 180,E1 -3310.892,E2 -3310.892} C_VEL
LIN {X 0,Y 552.597,Z 271.063,A -85,B 0,C 180,E1 -3313.563,E2 -3313.563} C_VEL
LIN {X 0,Y 552.33,Z 291.093,A -85,B 0,C 180,E1 -3316.386,E2 -3316.386} C_VEL
LIN {X 0,Y 552.281,Z 294.915,A -85,B 0,C 180,E1 -3316.923,E2 -3316.923} C_VEL
LIN {X 0,Y 553.153,Z 302.997,A -85,B 0,C 180,E1 -3317.084,E2 -3317.084} C_VEL
LIN {X 0,Y 552.982,Z 315.482,A -85,B 0,C 180,E1 -3317.384,E2 -3317.384} C_VEL
LIN {X 0,Y 552.843,Z 328.396,A -85,B 0,C 180,E1 -3317.847,E2 -3317.847} C_VEL
LIN {X 0,Y 552.683,Z 340.531,A -85,B 0,C 180,E1 -3318.441,E2 -3318.441} C_VEL
LIN {X 0,Y 552.486,Z 352.21,A -85,B 0,C 180,E1 -3319.187,E2 -3319.187} C_VEL
LIN {X 0,Y 552.301,Z 362.616,A -85,B 0,C 180,E1 -3320.017,E2 -3320.017} C_VEL
LIN {X 0,Y 552.131,Z 371.123,A -85,B 0,C 180,E1 -3320.846,E2 -3320.846} C_VEL
LIN {X 0,Y 552.012,Z 378.968,A -85,B 0,C 180,E1 -3321.766,E2 -3321.766} C_VEL
LIN {X 0,Y 551.888,Z 386.628,A -85,B 0,C 180,E1 -3322.869,E2 -3322.869} C_VEL
LIN {X 0,Y 551.867,Z 393.684,A -85,B 0,C 180,E1 -3324.154,E2 -3324.154} C_VEL
LIN {X 0,Y 551.725,Z 398.376,A -85,B 0,C 180,E1 -3325.252,E2 -3325.252} C_VEL
LIN {X 0,Y 551.75,Z 401.963,A -85,B 0,C 180,E1 -3326.349,E2 -3326.349} C_VEL
LIN {X 0,Y 551.723,Z 403.812,A -85,B 0,C 180,E1 -3327.08,E2 -3327.08} C_VEL
LIN {X 0,Y 551.645,Z 406.186,A -85,B 0,C 180,E1 -3328.541,E2 -3328.541} C_VEL
LIN {X 0,Y 551.64,Z 407,A -85,B 0,C 180,E1 -3330.001,E2 -3330.001} C_VEL
LIN {X 0,Y 551.645,Z 406.182,A -85,B 0,C 180,E1 -3331.461,E2 -3331.461} C_VEL
LIN {X 0,Y 551.724,Z 403.805,A -85,B 0,C 180,E1 -3332.922,E2 -3332.922} C_VEL
LIN {X 0,Y 551.764,Z 400.892,A -85,B 0,C 180,E1 -3334.018,E2 -3334.018} C_VEL
LIN {X 0,Y 551.724,Z 396.946,A -85,B 0,C 180,E1 -3335.117,E2 -3335.117} C_VEL
LIN {X 0,Y 551.825,Z 391.187,A -85,B 0,C 180,E1 -3336.342,E2 -3336.342} C_VEL
LIN {X 0,Y 551.927,Z 384.23,A -85,B 0,C 180,E1 -3337.5,E2 -3337.5} C_VEL
LIN {X 0,Y 552.079,Z 375.985,A -85,B 0,C 180,E1 -3338.603,E2 -3338.603} C_VEL
LIN {X 0,Y 552.201,Z 367.53,A -85,B 0,C 180,E1 -3339.524,E2 -3339.524} C_VEL
LIN {X 0,Y 552.423,Z 357.083,A -85,B 0,C 180,E1 -3340.446,E2 -3340.446} C_VEL
LIN {X 0,Y 552.588,Z 345.178,A -85,B 0,C 180,E1 -3341.286,E2 -3341.286} C_VEL
LIN {X 0,Y 552.784,Z 333.472,A -85,B 0,C 180,E1 -3341.924,E2 -3341.924} C_VEL
LIN {X 0,Y 552.957,Z 321.151,A -85,B 0,C 180,E1 -3342.432,E2 -3342.432} C_VEL
LIN {X 0,Y 553.074,Z 308.487,A -85,B 0,C 180,E1 -3342.803,E2 -3342.803} C_VEL
LIN {X 0,Y 552.926,Z 300.051,A -85,B 0,C 180,E1 -3342.97,E2 -3342.97} C_VEL
LIN {X 0,Y 552.282,Z 294.902,A -85,B 0,C 180,E1 -3343.079,E2 -3343.079} C_VEL
LIN {X 0,Y 552.506,Z 276.453,A -85,B 0,C 180,E1 -3345.683,E2 -3345.683} C_VEL
LIN {X 0,Y 552.743,Z 255.99,A -85,B 0,C 180,E1 -3348.535,E2 -3348.535} C_VEL
LIN {X 0,Y 552.987,Z 238.388,A -85,B 0,C 180,E1 -3351.042,E2 -3351.042} C_VEL
LIN {X 0,Y 553.294,Z 221.155,A -85,B 0,C 180,E1 -3353.545,E2 -3353.545} C_VEL
LIN {X 0,Y 553.714,Z 202.189,A -85,B 0,C 180,E1 -3356.375,E2 -3356.375} C_VEL
LIN {X 0,Y 554.19,Z 185.592,A -85,B 0,C 180,E1 -3358.951,E2 -3358.951} C_VEL
LIN {X 0,Y 553.582,Z 181.251,A -85,B 0,C 180,E1 -3359.679,E2 -3359.679} C_VEL
LIN {X 0,Y 552.106,Z 174.716,A -85,B 0,C 180,E1 -3360.875,E2 -3360.875} C_VEL
LIN {X 0,Y 552.099,Z 174.719,A -85,B 0,C 180,E1 -3363.188,E2 -3363.188} C_VEL
LIN {X 0,Y 552.074,Z 174.716,A -85,B 0,C 180,E1 -3365.845,E2 -3365.845} C_VEL
LIN {X 0,Y 552.118,Z 174.715,A -85,B 0,C 180,E1 -3368.59,E2 -3368.59} C_VEL
LIN {X 0,Y 552.126,Z 174.708,A -85,B 0,C 180,E1 -3371.446,E2 -3371.446} C_VEL
LIN {X 0,Y 552.093,Z 174.712,A -85,B 0,C 180,E1 -3374.531,E2 -3374.531} C_VEL
LIN {X 0,Y 552.135,Z 174.712,A -85,B 0,C 180,E1 -3377.585,E2 -3377.585} C_VEL
LIN {X 0,Y 552.13,Z 174.71,A -85,B 0,C 180,E1 -3380.473,E2 -3380.473} C_VEL
LIN {X 0,Y 552.101,Z 174.713,A -85,B 0,C 180,E1 -3383.319,E2 -3383.319} C_VEL
LIN {X 0,Y 552.048,Z 174.826,A -85,B 0,C 180,E1 -3386.043,E2 -3386.043} C_VEL
LIN {X 0,Y 552.049,Z 183.849,A -85,B 0,C 180,E1 -3388.536,E2 -3388.536} C_VEL
LIN {X 0,Y 552.084,Z 193.74,A -85,B 0,C 180,E1 -3391.447,E2 -3391.447} C_VEL
LIN {X 0,Y 552.138,Z 203.087,A -85,B 0,C 180,E1 -3394.356,E2 -3394.356} C_VEL
LIN {X 0,Y 552.092,Z 211.61,A -85,B 0,C 180,E1 -3397.154,E2 -3397.154} C_VEL
LIN {X 0,Y 552.065,Z 219.942,A -85,B 0,C 180,E1 -3399.896,E2 -3399.896} C_VEL
LIN {X 0,Y 551.962,Z 228.076,A -85,B 0,C 180,E1 -3402.739,E2 -3402.739} C_VEL
LIN {X 0,Y 551.912,Z 235.792,A -85,B 0,C 180,E1 -3405.417,E2 -3405.417} C_VEL
LIN {X 0,Y 551.883,Z 240.694,A -85,B 0,C 180,E1 -3407.065,E2 -3407.065} C_VEL
LIN {X 0,Y 553.073,Z 248.509,A -85,B 0,C 180,E1 -3407.245,E2 -3407.245} C_VEL
LIN {X 0,Y 552.956,Z 261.282,A -85,B 0,C 180,E1 -3407.615,E2 -3407.615} C_VEL
LIN {X 0,Y 552.722,Z 274.465,A -85,B 0,C 180,E1 -3408.169,E2 -3408.169} C_VEL
LIN {X 0,Y 552.594,Z 285.602,A -85,B 0,C 180,E1 -3408.786,E2 -3408.786} C_VEL
LIN {X 0,Y 552.399,Z 296.527,A -85,B 0,C 180,E1 -3409.555,E2 -3409.555} C_VEL
LIN {X 0,Y 552.226,Z 307.079,A -85,B 0,C 180,E1 -3410.477,E2 -3410.477} C_VEL
LIN {X 0,Y 552.084,Z 315.609,A -85,B 0,C 180,E1 -3411.398,E2 -3411.398} C_VEL
LIN {X 0,Y 551.928,Z 323.937,A -85,B 0,C 180,E1 -3412.5,E2 -3412.5} C_VEL
LIN {X 0,Y 551.813,Z 330.913,A -85,B 0,C 180,E1 -3413.65,E2 -3413.65} C_VEL
LIN {X 0,Y 551.803,Z 335.186,A -85,B 0,C 180,E1 -3414.519,E2 -3414.519} C_VEL
LIN {X 0,Y 551.768,Z 339.545,A -85,B 0,C 180,E1 -3415.617,E2 -3415.617} C_VEL
LIN {X 0,Y 551.751,Z 341.833,A -85,B 0,C 180,E1 -3416.348,E2 -3416.348} C_VEL
LIN {X 0,Y 551.724,Z 343.689,A -85,B 0,C 180,E1 -3417.079,E2 -3417.079} C_VEL
LIN {X 0,Y 551.656,Z 345.136,A -85,B 0,C 180,E1 -3417.81,E2 -3417.81} C_VEL
LIN {X 0,Y 551.643,Z 346.755,A -85,B 0,C 180,E1 -3419.27,E2 -3419.27} C_VEL
LIN {X 0,Y 551.641,Z 346.996,A -85,B 0,C 180,E1 -3420,E2 -3420} C_VEL
LIN {X 0,Y 551.641,Z 346.812,A -85,B 0,C 180,E1 -3420.73,E2 -3420.73} C_VEL
LIN {X 0,Y 551.655,Z 345.274,A -85,B 0,C 180,E1 -3422.19,E2 -3422.19} C_VEL
LIN {X 0,Y 551.724,Z 343.9,A -85,B 0,C 180,E1 -3422.921,E2 -3422.921} C_VEL
LIN {X 0,Y 551.764,Z 341.03,A -85,B 0,C 180,E1 -3424.017,E2 -3424.017} C_VEL
LIN {X 0,Y 551.724,Z 337.126,A -85,B 0,C 180,E1 -3425.116,E2 -3425.116} C_VEL
LIN {X 0,Y 551.811,Z 331.382,A -85,B 0,C 180,E1 -3426.349,E2 -3426.349} C_VEL
LIN {X 0,Y 551.926,Z 324.56,A -85,B 0,C 180,E1 -3427.5,E2 -3427.5} C_VEL
LIN {X 0,Y 552.063,Z 316.345,A -85,B 0,C 180,E1 -3428.603,E2 -3428.603} C_VEL
LIN {X 0,Y 552.197,Z 307.963,A -85,B 0,C 180,E1 -3429.524,E2 -3429.524} C_VEL
LIN {X 0,Y 552.381,Z 297.662,A -85,B 0,C 180,E1 -3430.446,E2 -3430.446} C_VEL
LIN {X 0,Y 552.549,Z 286.004,A -85,B 0,C 180,E1 -3431.279,E2 -3431.279} C_VEL
LIN {X 0,Y 552.75,Z 274.406,A -85,B 0,C 180,E1 -3431.924,E2 -3431.924} C_VEL
LIN {X 0,Y 552.927,Z 262.425,A -85,B 0,C 180,E1 -3432.432,E2 -3432.432} C_VEL
LIN {X 0,Y 553.073,Z 249.401,A -85,B 0,C 180,E1 -3432.825,E2 -3432.825} C_VEL
LIN {X 0,Y 551.804,Z 240.486,A -85,B 0,C 180,E1 -3433.043,E2 -3433.043} C_VEL
LIN {X 0,Y 551.878,Z 232.172,A -85,B 0,C 180,E1 -3435.89,E2 -3435.89} C_VEL
LIN {X 0,Y 551.994,Z 224.521,A -85,B 0,C 180,E1 -3438.56,E2 -3438.56} C_VEL
LIN {X 0,Y 552.069,Z 216.756,A -85,B 0,C 180,E1 -3441.273,E2 -3441.273} C_VEL
LIN {X 0,Y 552.124,Z 207.503,A -85,B 0,C 180,E1 -3444.437,E2 -3444.437} C_VEL
LIN {X 0,Y 552.184,Z 199.136,A -85,B 0,C 180,E1 -3447.271,E2 -3447.271} C_VEL
LIN {X 0,Y 552.174,Z 197.139,A -85,B 0,C 180,E1 -3447.951,E2 -3447.951} C_VEL
LIN {X 0,Y 551.526,Z 195.535,A -85,B 0,C 180,E1 -3448.536,E2 -3448.536} C_VEL
LIN {X 0,Y 548.76,Z 193.217,A -85,B 0,C 180,E1 -3449.497,E2 -3449.497} C_VEL
LIN {X 0,Y 546.414,Z 191.393,A -85,B 0,C 180,E1 -3450.272,E2 -3450.272} C_VEL
LIN {X 0,Y 545.388,Z 189.867,A -85,B 0,C 180,E1 -3450.864,E2 -3450.864} C_VEL
LIN {X 0,Y 545.294,Z 189.309,A -85,B 0,C 180,E1 -3451.064,E2 -3451.064} C_VEL
LIN {X 0,Y 545.287,Z 181.809,A -85,B 0,C 180,E1 -3453.657,E2 -3453.657} C_VEL
LIN {X 0,Y 545.233,Z 176.575,A -85,B 0,C 180,E1 -3455.454,E2 -3455.454} C_VEL
LIN {X 0,Y 545.065,Z 175.593,A -85,B 0,C 180,E1 -3455.851,E2 -3455.851} C_VEL
LIN {X 0,Y 545.105,Z 175.587,A -85,B 0,C 180,E1 -3459.323,E2 -3459.323} C_VEL
LIN {X 0,Y 545.07,Z 175.588,A -85,B 0,C 180,E1 -3462.104,E2 -3462.104} C_VEL
LIN {X 0,Y 545.034,Z 175.591,A -85,B 0,C 180,E1 -3465.17,E2 -3465.17} C_VEL
LIN {X 0,Y 545.083,Z 175.587,A -85,B 0,C 180,E1 -3467.897,E2 -3467.897} C_VEL
LIN {X 0,Y 545.083,Z 175.591,A -85,B 0,C 180,E1 -3470.818,E2 -3470.818} C_VEL
LIN {X 0,Y 545.018,Z 175.597,A -85,B 0,C 180,E1 -3473.617,E2 -3473.617} C_VEL
LIN {X 0,Y 545.052,Z 175.59,A -85,B 0,C 180,E1 -3476.326,E2 -3476.326} C_VEL
LIN {X 0,Y 545.061,Z 175.593,A -85,B 0,C 180,E1 -3478.951,E2 -3478.951} C_VEL
LIN {X 0,Y 544.939,Z 175.609,A -85,B 0,C 180,E1 -3480.653,E2 -3480.653} C_VEL
LIN {X 0,Y 544.963,Z 176.335,A -85,B 0,C 180,E1 -3481.499,E2 -3481.499} C_VEL
LIN {X 0,Y 544.916,Z 180.343,A -85,B 0,C 180,E1 -3484.532,E2 -3484.532} C_VEL
LIN {X 0,Y 544.826,Z 183.806,A -85,B 0,C 180,E1 -3487.232,E2 -3487.232} C_VEL
LIN {X 0,Y 544.785,Z 187.943,A -85,B 0,C 180,E1 -3490.402,E2 -3490.402} C_VEL
LIN {X 0,Y 544.705,Z 192.114,A -85,B 0,C 180,E1 -3493.509,E2 -3493.509} C_VEL
LIN {X 0,Y 544.715,Z 195.312,A -85,B 0,C 180,E1 -3495.809,E2 -3495.809} C_VEL
LIN {X 0,Y 544.696,Z 199.433,A -85,B 0,C 180,E1 -3498.84,E2 -3498.84} C_VEL
LIN {X 0,Y 544.615,Z 204.334,A -85,B 0,C 180,E1 -3502.305,E2 -3502.305} C_VEL
LIN {X 0,Y 544.794,Z 205.377,A -85,B 0,C 180,E1 -3502.377,E2 -3502.377} C_VEL
LIN {X 0,Y 545.247,Z 211.937,A -85,B 0,C 180,E1 -3502.64,E2 -3502.64} C_VEL
LIN {X 0,Y 545.166,Z 219.793,A -85,B 0,C 180,E1 -3503.049,E2 -3503.049} C_VEL
LIN {X 0,Y 545.078,Z 227.071,A -85,B 0,C 180,E1 -3503.542,E2 -3503.542} C_VEL
LIN {X 0,Y 544.945,Z 235.174,A -85,B 0,C 180,E1 -3504.263,E2 -3504.263} C_VEL
LIN {X 0,Y 544.969,Z 241.48,A -85,B 0,C 180,E1 -3505.005,E2 -3505.005} C_VEL
LIN {X 0,Y 544.85,Z 247.507,A -85,B 0,C 180,E1 -3505.931,E2 -3505.931} C_VEL
LIN {X 0,Y 544.756,Z 252.61,A -85,B 0,C 180,E1 -3507.041,E2 -3507.041} C_VEL
LIN {X 0,Y 544.67,Z 255.008,A -85,B 0,C 180,E1 -3507.781,E2 -3507.781} C_VEL
LIN {X 0,Y 544.651,Z 256.666,A -85,B 0,C 180,E1 -3508.52,E2 -3508.52} C_VEL
LIN {X 0,Y 544.635,Z 257.641,A -85,B 0,C 180,E1 -3509.26,E2 -3509.26} C_VEL
LIN {X 0,Y 544.63,Z 257.99,A -85,B 0,C 180,E1 -3509.999,E2 -3509.999} C_VEL
LIN {X 0,Y 544.634,Z 257.736,A -85,B 0,C 180,E1 -3510.738,E2 -3510.738} C_VEL
LIN {X 0,Y 544.626,Z 256.84,A -85,B 0,C 180,E1 -3511.478,E2 -3511.478} C_VEL
LIN {X 0,Y 544.728,Z 254.181,A -85,B 0,C 180,E1 -3512.587,E2 -3512.587} C_VEL
LIN {X 0,Y 544.781,Z 251.517,A -85,B 0,C 180,E1 -3513.327,E2 -3513.327} C_VEL
LIN {X 0,Y 544.846,Z 246.968,A -85,B 0,C 180,E1 -3514.253,E2 -3514.253} C_VEL
LIN {X 0,Y 544.947,Z 242.14,A -85,B 0,C 180,E1 -3514.993,E2 -3514.993} C_VEL
LIN {X 0,Y 544.938,Z 236.052,A -85,B 0,C 180,E1 -3515.735,E2 -3515.735} C_VEL
LIN {X 0,Y 545.059,Z 229.311,A -85,B 0,C 180,E1 -3516.371,E2 -3516.371} C_VEL
LIN {X 0,Y 545.104,Z 221.025,A -85,B 0,C 180,E1 -3516.971,E2 -3516.971} C_VEL
LIN {X 0,Y 545.268,Z 211.905,A -85,B 0,C 180,E1 -3517.451,E2 -3517.451} C_VEL
LIN {X 0,Y 544.719,Z 205.003,A -85,B 0,C 180,E1 -3517.727,E2 -3517.727} C_VEL
LIN {X 0,Y 544.62,Z 204.344,A -85,B 0,C 180,E1 -3517.786,E2 -3517.786} C_VEL
LIN {X 0,Y 544.706,Z 199.403,A -85,B 0,C 180,E1 -3521.308,E2 -3521.308} C_VEL
LIN {X 0,Y 544.707,Z 194.831,A -85,B 0,C 180,E1 -3524.606,E2 -3524.606} C_VEL
LIN {X 0,Y 544.718,Z 191.153,A -85,B 0,C 180,E1 -3527.3,E2 -3527.3} C_VEL
LIN {X 0,Y 544.767,Z 187.038,A -85,B 0,C 180,E1 -3530.384,E2 -3530.384} C_VEL
LIN {X 0,Y 544.816,Z 183.948,A -85,B 0,C 180,E1 -3532.766,E2 -3532.766} C_VEL
LIN {X 0,Y 544.909,Z 180.498,A -85,B 0,C 180,E1 -3535.467,E2 -3535.467} C_VEL
LIN {X 0,Y 544.957,Z 176.471,A -85,B 0,C 180,E1 -3538.499,E2 -3538.499} C_VEL
LIN {X 0,Y 544.946,Z 175.609,A -85,B 0,C 180,E1 -3539.344,E2 -3539.344} C_VEL
LIN {X 0,Y 545.051,Z 175.592,A -85,B 0,C 180,E1 -3541.914,E2 -3541.914} C_VEL
LIN {X 0,Y 545.072,Z 175.585,A -85,B 0,C 180,E1 -3544.562,E2 -3544.562} C_VEL
LIN {X 0,Y 545.033,Z 175.597,A -85,B 0,C 180,E1 -3547.303,E2 -3547.303} C_VEL
LIN {X 0,Y 545.065,Z 175.585,A -85,B 0,C 180,E1 -3550.141,E2 -3550.141} C_VEL
LIN {X 0,Y 545.08,Z 175.592,A -85,B 0,C 180,E1 -3553.105,E2 -3553.105} C_VEL
LIN {X 0,Y 545.051,Z 175.587,A -85,B 0,C 180,E1 -3556.224,E2 -3556.224} C_VEL
LIN {X 0,Y 545.09,Z 175.589,A -85,B 0,C 180,E1 -3558.886,E2 -3558.886} C_VEL
LIN {X 0,Y 545.046,Z 175.587,A -85,B 0,C 180,E1 -3561.762,E2 -3561.762} C_VEL
LIN {X 0,Y 545.058,Z 175.594,A -85,B 0,C 180,E1 -3564.533,E2 -3564.533} C_VEL
LIN {X 0,Y 545.075,Z 175.584,A -85,B 0,C 180,E1 -3567.212,E2 -3567.212} C_VEL
LIN {X 0,Y 545.093,Z 175.583,A -85,B 0,C 180,E1 -3569.812,E2 -3569.812} C_VEL
LIN {X 0,Y 545.092,Z 175.583,A -85,B 0,C 180,E1 -3572.824,E2 -3572.824} C_VEL
LIN {X 0,Y 545.043,Z 175.588,A -85,B 0,C 180,E1 -3575.63,E2 -3575.63} C_VEL
LIN {X 0,Y 545.059,Z 175.584,A -85,B 0,C 180,E1 -3578.836,E2 -3578.836} C_VEL
LIN {X 0,Y 545.074,Z 175.584,A -85,B 0,C 180,E1 -3581.195,E2 -3581.195} C_VEL
LIN {X 0,Y 545.068,Z 175.59,A -85,B 0,C 180,E1 -3583.521,E2 -3583.521} C_VEL
LIN {X 0,Y 545.085,Z 175.588,A -85,B 0,C 180,E1 -3585.82,E2 -3585.82} C_VEL
LIN {X 0,Y 545.121,Z 175.578,A -85,B 0,C 180,E1 -3588.849,E2 -3588.849} C_VEL
LIN {X 0,Y 545.124,Z 175.579,A -85,B 0,C 180,E1 -3591.847,E2 -3591.847} C_VEL
LIN {X 0,Y 545.195,Z 175.571,A -85,B 0,C 180,E1 -3594.823,E2 -3594.823} C_VEL
LIN {X 0,Y 545.177,Z 175.571,A -85,B 0,C 180,E1 -3597.784,E2 -3597.784} C_VEL
LIN {X 0,Y 545.206,Z 175.57,A -85,B 0,C 180,E1 -3600.739,E2 -3600.739} C_VEL
LIN {X 0,Y 545.16,Z 175.579,A -85,B 0,C 180,E1 -3602.956,E2 -3602.956} C_VEL
LIN {X 0,Y 545.149,Z 175.574,A -85,B 0,C 180,E1 -3605.92,E2 -3605.92} C_VEL
LIN {X 0,Y 545.099,Z 175.583,A -85,B 0,C 180,E1 -3608.9,E2 -3608.9} C_VEL
LIN {X 0,Y 545.091,Z 175.584,A -85,B 0,C 180,E1 -3611.905,E2 -3611.905} C_VEL
LIN {X 0,Y 545.071,Z 175.585,A -85,B 0,C 180,E1 -3614.944,E2 -3614.944} C_VEL
LIN {X 0,Y 545.044,Z 175.593,A -85,B 0,C 180,E1 -3618.027,E2 -3618.027} C_VEL
LIN {X 0,Y 545.077,Z 175.588,A -85,B 0,C 180,E1 -3620.373,E2 -3620.373} C_VEL
LIN {X 0,Y 545.059,Z 175.59,A -85,B 0,C 180,E1 -3623.56,E2 -3623.56} C_VEL
LIN {X 0,Y 545.027,Z 175.596,A -85,B 0,C 180,E1 -3626.003,E2 -3626.003} C_VEL
LIN {X 0,Y 545.006,Z 175.593,A -85,B 0,C 180,E1 -3628.735,E2 -3628.735} C_VEL
LIN {X 0,Y 545.05,Z 175.589,A -85,B 0,C 180,E1 -3631.049,E2 -3631.049} C_VEL
LIN {X 0,Y 545.051,Z 175.591,A -85,B 0,C 180,E1 -3633.673,E2 -3633.673} C_VEL
LIN {X 0,Y 545.054,Z 175.591,A -85,B 0,C 180,E1 -3636.926,E2 -3636.926} C_VEL
LIN {X 0,Y 545.054,Z 175.585,A -85,B 0,C 180,E1 -3640.144,E2 -3640.144} C_VEL
LIN {X 0,Y 545.037,Z 175.596,A -85,B 0,C 180,E1 -3643.111,E2 -3643.111} C_VEL
LIN {X 0,Y 545.041,Z 175.59,A -85,B 0,C 180,E1 -3646.227,E2 -3646.227} C_VEL
LIN {X 0,Y 545.074,Z 175.592,A -85,B 0,C 180,E1 -3648.886,E2 -3648.886} C_VEL
LIN {X 0,Y 545.076,Z 175.589,A -85,B 0,C 180,E1 -3650.82,E2 -3650.82} C_VEL
LIN {X 0,Y 545.037,Z 175.589,A -85,B 0,C 180,E1 -3653.621,E2 -3653.621} C_VEL
LIN {X 0,Y 545.062,Z 175.594,A -85,B 0,C 180,E1 -3656.329,E2 -3656.329} C_VEL
LIN {X 0,Y 545.104,Z 175.609,A -85,B 0,C 180,E1 -3658.855,E2 -3658.855} C_VEL
LIN {X 0,Y 547.184,Z 184.939,A -85,B 0,C 180,E1 -3660.577,E2 -3660.577} C_VEL
LIN {X 0,Y 547.148,Z 192.766,A -85,B 0,C 180,E1 -3661.855,E2 -3661.855} C_VEL
LIN {X 0,Y 546.622,Z 211.196,A -85,B 0,C 180,E1 -3664.696,E2 -3664.696} C_VEL
LIN {X 0,Y 546.207,Z 231.18,A -85,B 0,C 180,E1 -3667.685,E2 -3667.685} C_VEL
LIN {X 0,Y 545.84,Z 250.076,A -85,B 0,C 180,E1 -3670.443,E2 -3670.443} C_VEL
LIN {X 0,Y 545.575,Z 270.41,A -85,B 0,C 180,E1 -3673.345,E2 -3673.345} C_VEL
LIN {X 0,Y 545.299,Z 292.334,A -85,B 0,C 180,E1 -3676.397,E2 -3676.397} C_VEL
LIN {X 0,Y 545.281,Z 295.209,A -85,B 0,C 180,E1 -3676.776,E2 -3676.776} C_VEL
LIN {X 0,Y 546.237,Z 302.997,A -85,B 0,C 180,E1 -3676.918,E2 -3676.918} C_VEL
LIN {X 0,Y 546.078,Z 315.48,A -85,B 0,C 180,E1 -3677.221,E2 -3677.221} C_VEL
LIN {X 0,Y 545.892,Z 328.386,A -85,B 0,C 180,E1 -3677.689,E2 -3677.689} C_VEL
LIN {X 0,Y 545.764,Z 339.271,A -85,B 0,C 180,E1 -3678.222,E2 -3678.222} C_VEL
LIN {X 0,Y 545.565,Z 349.607,A -85,B 0,C 180,E1 -3678.86,E2 -3678.86} C_VEL
LIN {X 0,Y 545.316,Z 360.478,A -85,B 0,C 180,E1 -3679.7,E2 -3679.7} C_VEL
LIN {X 0,Y 545.141,Z 369.343,A -85,B 0,C 180,E1 -3680.54,E2 -3680.54} C_VEL
LIN {X 0,Y 544.977,Z 378.968,A -85,B 0,C 180,E1 -3681.659,E2 -3681.659} C_VEL
LIN {X 0,Y 544.822,Z 386.628,A -85,B 0,C 180,E1 -3682.776,E2 -3682.776} C_VEL
LIN {X 0,Y 544.776,Z 393.683,A -85,B 0,C 180,E1 -3684.077,E2 -3684.077} C_VEL
LIN {X 0,Y 544.628,Z 398.376,A -85,B 0,C 180,E1 -3685.19,E2 -3685.19} C_VEL
LIN {X 0,Y 544.669,Z 401.963,A -85,B 0,C 180,E1 -3686.302,E2 -3686.302} C_VEL
LIN {X 0,Y 544.65,Z 403.812,A -85,B 0,C 180,E1 -3687.042,E2 -3687.042} C_VEL
LIN {X 0,Y 544.546,Z 406.185,A -85,B 0,C 180,E1 -3688.522,E2 -3688.522} C_VEL
LIN {X 0,Y 544.541,Z 407,A -85,B 0,C 180,E1 -3690.001,E2 -3690.001} C_VEL
LIN {X 0,Y 544.546,Z 406.182,A -85,B 0,C 180,E1 -3691.48,E2 -3691.48} C_VEL
LIN {X 0,Y 544.651,Z 403.805,A -85,B 0,C 180,E1 -3692.96,E2 -3692.96} C_VEL
LIN {X 0,Y 544.684,Z 400.892,A -85,B 0,C 180,E1 -3694.07,E2 -3694.07} C_VEL
LIN {X 0,Y 544.654,Z 396.946,A -85,B 0,C 180,E1 -3695.183,E2 -3695.183} C_VEL
LIN {X 0,Y 544.737,Z 391.593,A -85,B 0,C 180,E1 -3696.349,E2 -3696.349} C_VEL
LIN {X 0,Y 544.86,Z 384.229,A -85,B 0,C 180,E1 -3697.598,E2 -3697.598} C_VEL
LIN {X 0,Y 545.027,Z 375.985,A -85,B 0,C 180,E1 -3698.716,E2 -3698.716} C_VEL
LIN {X 0,Y 545.165,Z 367.531,A -85,B 0,C 180,E1 -3699.649,E2 -3699.649} C_VEL
LIN {X 0,Y 545.415,Z 357.081,A -85,B 0,C 180,E1 -3700.582,E2 -3700.582} C_VEL
LIN {X 0,Y 545.611,Z 345.577,A -85,B 0,C 180,E1 -3701.406,E2 -3701.406} C_VEL
LIN {X 0,Y 545.799,Z 335.39,A -85,B 0,C 180,E1 -3701.985,E2 -3701.985} C_VEL
LIN {X 0,Y 545.97,Z 323.751,A -85,B 0,C 180,E1 -3702.5,E2 -3702.5} C_VEL
LIN {X 0,Y 546.139,Z 310.318,A -85,B 0,C 180,E1 -3702.921,E2 -3702.921} C_VEL
LIN {X 0,Y 546.134,Z 301.555,A -85,B 0,C 180,E1 -3703.11,E2 -3703.11} C_VEL
LIN {X 0,Y 545.264,Z 294.87,A -85,B 0,C 180,E1 -3703.25,E2 -3703.25} C_VEL
LIN {X 0,Y 545.474,Z 274.444,A -85,B 0,C 180,E1 -3706.083,E2 -3706.083} C_VEL
LIN {X 0,Y 545.747,Z 254.075,A -85,B 0,C 180,E1 -3708.976,E2 -3708.976} C_VEL
LIN {X 0,Y 546.059,Z 237.946,A -85,B 0,C 180,E1 -3711.322,E2 -3711.322} C_VEL
LIN {X 0,Y 546.428,Z 219.523,A -85,B 0,C 180,E1 -3714.051,E2 -3714.051} C_VEL
LIN {X 0,Y 546.859,Z 201.883,A -85,B 0,C 180,E1 -3716.732,E2 -3716.732} C_VEL
LIN {X 0,Y 547.306,Z 186.448,A -85,B 0,C 180,E1 -3719.168,E2 -3719.168} C_VEL
LIN {X 0,Y 545.652,Z 178.225,A -85,B 0,C 180,E1 -3720.649,E2 -3720.649} C_VEL
LIN {X 0,Y 545.087,Z 175.591,A -85,B 0,C 180,E1 -3721.174,E2 -3721.174} C_VEL
LIN {X 0,Y 545.046,Z 175.595,A -85,B 0,C 180,E1 -3723.674,E2 -3723.674} C_VEL
LIN {X 0,Y 545.069,Z 175.592,A -85,B 0,C 180,E1 -3726.925,E2 -3726.925} C_VEL
LIN {X 0,Y 545.069,Z 175.592,A -85,B 0,C 180,E1 -3730.143,E2 -3730.143} C_VEL
LIN {X 0,Y 545.084,Z 175.585,A -85,B 0,C 180,E1 -3733.107,E2 -3733.107} C_VEL
LIN {X 0,Y 545.054,Z 175.589,A -85,B 0,C 180,E1 -3736.227,E2 -3736.227} C_VEL
LIN {X 0,Y 545.085,Z 175.589,A -85,B 0,C 180,E1 -3738.886,E2 -3738.886} C_VEL
LIN {X 0,Y 545.048,Z 175.59,A -85,B 0,C 180,E1 -3741.865,E2 -3741.865} C_VEL
LIN {X 0,Y 545.023,Z 175.6,A -85,B 0,C 180,E1 -3744.53,E2 -3744.53} C_VEL
LIN {X 0,Y 545.024,Z 175.701,A -85,B 0,C 180,E1 -3745.992,E2 -3745.992} C_VEL
LIN {X 0,Y 545.028,Z 185.219,A -85,B 0,C 180,E1 -3748.641,E2 -3748.641} C_VEL
LIN {X 0,Y 545.043,Z 194.865,A -85,B 0,C 180,E1 -3751.504,E2 -3751.504} C_VEL
LIN {X 0,Y 545.078,Z 204.413,A -85,B 0,C 180,E1 -3754.496,E2 -3754.496} C_VEL
LIN {X 0,Y 545.042,Z 212.819,A -85,B 0,C 180,E1 -3757.242,E2 -3757.242} C_VEL
LIN {X 0,Y 545.019,Z 221.881,A -85,B 0,C 180,E1 -3760.278,E2 -3760.278} C_VEL
LIN {X 0,Y 544.916,Z 230.149,A -85,B 0,C 180,E1 -3763.131,E2 -3763.131} C_VEL
LIN {X 0,Y 544.848,Z 237.815,A -85,B 0,C 180,E1 -3765.813,E2 -3765.813} C_VEL
LIN {X 0,Y 544.813,Z 240.856,A -85,B 0,C 180,E1 -3766.894,E2 -3766.894} C_VEL
LIN {X 0,Y 546.143,Z 249.561,A -85,B 0,C 180,E1 -3767.104,E2 -3767.104} C_VEL
LIN {X 0,Y 545.997,Z 262.606,A -85,B 0,C 180,E1 -3767.502,E2 -3767.502} C_VEL
LIN {X 0,Y 545.787,Z 274.537,A -85,B 0,C 180,E1 -3768.016,E2 -3768.016} C_VEL
LIN {X 0,Y 545.612,Z 285.967,A -85,B 0,C 180,E1 -3768.66,E2 -3768.66} C_VEL
LIN {X 0,Y 545.389,Z 297.711,A -85,B 0,C 180,E1 -3769.513,E2 -3769.513} C_VEL
LIN {X 0,Y 545.207,Z 307.087,A -85,B 0,C 180,E1 -3770.353,E2 -3770.353} C_VEL
LIN {X 0,Y 545.041,Z 315.613,A -85,B 0,C 180,E1 -3771.286,E2 -3771.286} C_VEL
LIN {X 0,Y 544.861,Z 323.938,A -85,B 0,C 180,E1 -3772.403,E2 -3772.403} C_VEL
LIN {X 0,Y 544.754,Z 330.08,A -85,B 0,C 180,E1 -3773.414,E2 -3773.414} C_VEL
LIN {X 0,Y 544.74,Z 335.187,A -85,B 0,C 180,E1 -3774.447,E2 -3774.447} C_VEL
LIN {X 0,Y 544.666,Z 339.548,A -85,B 0,C 180,E1 -3775.56,E2 -3775.56} C_VEL
LIN {X 0,Y 544.669,Z 341.833,A -85,B 0,C 180,E1 -3776.301,E2 -3776.301} C_VEL
LIN {X 0,Y 544.651,Z 343.688,A -85,B 0,C 180,E1 -3777.041,E2 -3777.041} C_VEL
LIN {X 0,Y 544.571,Z 345.137,A -85,B 0,C 180,E1 -3777.781,E2 -3777.781} C_VEL
LIN {X 0,Y 544.543,Z 346.755,A -85,B 0,C 180,E1 -3779.261,E2 -3779.261} C_VEL
LIN {X 0,Y 544.541,Z 346.996,A -85,B 0,C 180,E1 -3780,E2 -3780} C_VEL
LIN {X 0,Y 544.542,Z 346.811,A -85,B 0,C 180,E1 -3780.74,E2 -3780.74} C_VEL
LIN {X 0,Y 544.57,Z 345.274,A -85,B 0,C 180,E1 -3782.219,E2 -3782.219} C_VEL
LIN {X 0,Y 544.651,Z 343.897,A -85,B 0,C 180,E1 -3782.959,E2 -3782.959} C_VEL
LIN {X 0,Y 544.684,Z 341.026,A -85,B 0,C 180,E1 -3784.07,E2 -3784.07} C_VEL
LIN {X 0,Y 544.653,Z 337.121,A -85,B 0,C 180,E1 -3785.182,E2 -3785.182} C_VEL
LIN {X 0,Y 544.724,Z 331.877,A -85,B 0,C 180,E1 -3786.335,E2 -3786.335} C_VEL
LIN {X 0,Y 544.836,Z 325.737,A -85,B 0,C 180,E1 -3787.411,E2 -3787.411} C_VEL
LIN {X 0,Y 544.994,Z 317.858,A -85,B 0,C 180,E1 -3788.528,E2 -3788.528} C_VEL
LIN {X 0,Y 545.159,Z 307.954,A -85,B 0,C 180,E1 -3789.648,E2 -3789.648} C_VEL
LIN {X 0,Y 545.374,Z 297.659,A -85,B 0,C 180,E1 -3790.582,E2 -3790.582} C_VEL
LIN {X 0,Y 545.571,Z 286.42,A -85,B 0,C 180,E1 -3791.399,E2 -3791.399} C_VEL
LIN {X 0,Y 545.767,Z 276.32,A -85,B 0,C 180,E1 -3791.985,E2 -3791.985} C_VEL
LIN {X 0,Y 545.972,Z 263.695,A -85,B 0,C 180,E1 -3792.546,E2 -3792.546} C_VEL
LIN {X 0,Y 546.138,Z 250.378,A -85,B 0,C 180,E1 -3792.967,E2 -3792.967} C_VEL
LIN {X 0,Y 544.745,Z 240.599,A -85,B 0,C 180,E1 -3793.215,E2 -3793.215} C_VEL
LIN {X 0,Y 544.843,Z 232.309,A -85,B 0,C 180,E1 -3796.101,E2 -3796.101} C_VEL
LIN {X 0,Y 544.939,Z 224.661,A -85,B 0,C 180,E1 -3798.81,E2 -3798.81} C_VEL
LIN {X 0,Y 545.05,Z 216.008,A -85,B 0,C 180,E1 -3801.815,E2 -3801.815} C_VEL
LIN {X 0,Y 545.091,Z 207.457,A -85,B 0,C 180,E1 -3804.774,E2 -3804.774} C_VEL
LIN {X 0,Y 545.184,Z 199.08,A -85,B 0,C 180,E1 -3807.651,E2 -3807.651} C_VEL
LIN {X 0,Y 545.272,Z 190.587,A -85,B 0,C 180,E1 -3810.613,E2 -3810.613} C_VEL
LIN {X 0,Y 545.294,Z 189.309,A -85,B 0,C 180,E1 -3811.064,E2 -3811.064} C_VEL
LIN {X 0,Y 544.595,Z 187.715,A -85,B 0,C 180,E1 -3811.657,E2 -3811.657} C_VEL
LIN {X 0,Y 541.724,Z 185.356,A -85,B 0,C 180,E1 -3812.628,E2 -3812.628} C_VEL
LIN {X 0,Y 539.342,Z 183.487,A -85,B 0,C 180,E1 -3813.41,E2 -3813.41} C_VEL
LIN {X 0,Y 538.352,Z 181.919,A -85,B 0,C 180,E1 -3814.01,E2 -3814.01} C_VEL
LIN {X 0,Y 538.288,Z 181.346,A -85,B 0,C 180,E1 -3814.211,E2 -3814.211} C_VEL
LIN {X 0,Y 538.228,Z 177.656,A -85,B 0,C 180,E1 -3815.484,E2 -3815.484} C_VEL
LIN {X 0,Y 538.039,Z 176.468,A -85,B 0,C 180,E1 -3815.917,E2 -3815.917} C_VEL
LIN {X 0,Y 538.015,Z 176.466,A -85,B 0,C 180,E1 -3818.831,E2 -3818.831} C_VEL
LIN {X 0,Y 538.029,Z 176.464,A -85,B 0,C 180,E1 -3821.774,E2 -3821.774} C_VEL
LIN {X 0,Y 538.003,Z 176.467,A -85,B 0,C 180,E1 -3824.863,E2 -3824.863} C_VEL
LIN {X 0,Y 538.024,Z 176.467,A -85,B 0,C 180,E1 -3827.214,E2 -3827.214} C_VEL
LIN {X 0,Y 538.027,Z 176.465,A -85,B 0,C 180,E1 -3830.203,E2 -3830.203} C_VEL
LIN {X 0,Y 537.976,Z 176.472,A -85,B 0,C 180,E1 -3833.062,E2 -3833.062} C_VEL
LIN {X 0,Y 538.003,Z 176.471,A -85,B 0,C 180,E1 -3835.825,E2 -3835.825} C_VEL
LIN {X 0,Y 538.012,Z 176.47,A -85,B 0,C 180,E1 -3838.498,E2 -3838.498} C_VEL
LIN {X 0,Y 537.878,Z 176.57,A -85,B 0,C 180,E1 -3841.097,E2 -3841.097} C_VEL
LIN {X 0,Y 537.881,Z 179.93,A -85,B 0,C 180,E1 -3843.624,E2 -3843.624} C_VEL
LIN {X 0,Y 537.812,Z 183.189,A -85,B 0,C 180,E1 -3846.17,E2 -3846.17} C_VEL
LIN {X 0,Y 537.726,Z 187.26,A -85,B 0,C 180,E1 -3849.335,E2 -3849.335} C_VEL
LIN {X 0,Y 537.674,Z 190.386,A -85,B 0,C 180,E1 -3851.716,E2 -3851.716} C_VEL
LIN {X 0,Y 537.634,Z 194.642,A -85,B 0,C 180,E1 -3854.844,E2 -3854.844} C_VEL
LIN {X 0,Y 537.608,Z 198.865,A -85,B 0,C 180,E1 -3857.926,E2 -3857.926} C_VEL
LIN {X 0,Y 537.548,Z 202.134,A -85,B 0,C 180,E1 -3860.213,E2 -3860.213} C_VEL
LIN {X 0,Y 537.575,Z 204.937,A -85,B 0,C 180,E1 -3862.18,E2 -3862.18} C_VEL
LIN {X 0,Y 538.345,Z 211.652,A -85,B 0,C 180,E1 -3862.451,E2 -3862.451} C_VEL
LIN {X 0,Y 538.234,Z 220.815,A -85,B 0,C 180,E1 -3862.92,E2 -3862.92} C_VEL
LIN {X 0,Y 538.143,Z 228.614,A -85,B 0,C 180,E1 -3863.463,E2 -3863.463} C_VEL
LIN {X 0,Y 538.01,Z 236.532,A -85,B 0,C 180,E1 -3864.189,E2 -3864.189} C_VEL
LIN {X 0,Y 538.013,Z 242.761,A -85,B 0,C 180,E1 -3864.94,E2 -3864.94} C_VEL
LIN {X 0,Y 537.868,Z 248.663,A -85,B 0,C 180,E1 -3865.878,E2 -3865.878} C_VEL
LIN {X 0,Y 537.769,Z 253.681,A -85,B 0,C 180,E1 -3867.003,E2 -3867.003} C_VEL
LIN {X 0,Y 537.664,Z 256.033,A -85,B 0,C 180,E1 -3867.752,E2 -3867.752} C_VEL
LIN {X 0,Y 537.651,Z 257.666,A -85,B 0,C 180,E1 -3868.501,E2 -3868.501} C_VEL
LIN {X 0,Y 537.625,Z 258.645,A -85,B 0,C 180,E1 -3869.25,E2 -3869.25} C_VEL
LIN {X 0,Y 537.617,Z 258.995,A -85,B 0,C 180,E1 -3869.999,E2 -3869.999} C_VEL
LIN {X 0,Y 537.624,Z 258.726,A -85,B 0,C 180,E1 -3870.748,E2 -3870.748} C_VEL
LIN {X 0,Y 537.603,Z 257.836,A -85,B 0,C 180,E1 -3871.497,E2 -3871.497} C_VEL
LIN {X 0,Y 537.734,Z 255.238,A -85,B 0,C 180,E1 -3872.621,E2 -3872.621} C_VEL
LIN {X 0,Y 537.806,Z 250.982,A -85,B 0,C 180,E1 -3873.745,E2 -3873.745} C_VEL
LIN {X 0,Y 537.936,Z 245.912,A -85,B 0,C 180,E1 -3874.683,E2 -3874.683} C_VEL
LIN {X 0,Y 537.989,Z 239.003,A -85,B 0,C 180,E1 -3875.622,E2 -3875.622} C_VEL
LIN {X 0,Y 538.081,Z 232.478,A -85,B 0,C 180,E1 -3876.297,E2 -3876.297} C_VEL
LIN {X 0,Y 538.191,Z 224.514,A -85,B 0,C 180,E1 -3876.937,E2 -3876.937} C_VEL
LIN {X 0,Y 538.292,Z 216.65,A -85,B 0,C 180,E1 -3877.407,E2 -3877.407} C_VEL
LIN {X 0,Y 538.266,Z 209.293,A -85,B 0,C 180,E1 -3877.737,E2 -3877.737} C_VEL
LIN {X 0,Y 537.562,Z 204.937,A -85,B 0,C 180,E1 -3877.913,E2 -3877.913} C_VEL
LIN {X 0,Y 537.659,Z 200.034,A -85,B 0,C 180,E1 -3881.373,E2 -3881.373} C_VEL
LIN {X 0,Y 537.643,Z 195.413,A -85,B 0,C 180,E1 -3884.687,E2 -3884.687} C_VEL
LIN {X 0,Y 537.676,Z 191.58,A -85,B 0,C 180,E1 -3887.495,E2 -3887.495} C_VEL
LIN {X 0,Y 537.725,Z 187.389,A -85,B 0,C 180,E1 -3890.663,E2 -3890.663} C_VEL
LIN {X 0,Y 537.808,Z 183.258,A -85,B 0,C 180,E1 -3893.896,E2 -3893.896} C_VEL
LIN {X 0,Y 537.867,Z 180.072,A -85,B 0,C 180,E1 -3896.375,E2 -3896.375} C_VEL
LIN {X 0,Y 537.902,Z 176.684,A -85,B 0,C 180,E1 -3898.908,E2 -3898.908} C_VEL
LIN {X 0,Y 538.002,Z 176.472,A -85,B 0,C 180,E1 -3901.5,E2 -3901.5} C_VEL
LIN {X 0,Y 538.019,Z 176.464,A -85,B 0,C 180,E1 -3904.172,E2 -3904.172} C_VEL
LIN {X 0,Y 538.001,Z 176.471,A -85,B 0,C 180,E1 -3907.169,E2 -3907.169} C_VEL
LIN {X 0,Y 538.021,Z 176.465,A -85,B 0,C 180,E1 -3909.795,E2 -3909.795} C_VEL
LIN {X 0,Y 538.017,Z 176.467,A -85,B 0,C 180,E1 -3912.784,E2 -3912.784} C_VEL
LIN {X 0,Y 538.026,Z 176.469,A -85,B 0,C 180,E1 -3915.14,E2 -3915.14} C_VEL
LIN {X 0,Y 538.034,Z 176.462,A -85,B 0,C 180,E1 -3918.227,E2 -3918.227} C_VEL
LIN {X 0,Y 538.008,Z 176.467,A -85,B 0,C 180,E1 -3921.169,E2 -3921.169} C_VEL
LIN {X 0,Y 538.022,Z 176.464,A -85,B 0,C 180,E1 -3924.082,E2 -3924.082} C_VEL
LIN {X 0,Y 538.028,Z 176.467,A -85,B 0,C 180,E1 -3926.727,E2 -3926.727} C_VEL
LIN {X 0,Y 538.029,Z 176.461,A -85,B 0,C 180,E1 -3929.553,E2 -3929.553} C_VEL
LIN {X 0,Y 538.04,Z 176.464,A -85,B 0,C 180,E1 -3931.95,E2 -3931.95} C_VEL
LIN {X 0,Y 538.067,Z 176.458,A -85,B 0,C 180,E1 -3934.467,E2 -3934.467} C_VEL
LIN {X 0,Y 538.014,Z 176.463,A -85,B 0,C 180,E1 -3936.928,E2 -3936.928} C_VEL
LIN {X 0,Y 538.068,Z 176.46,A -85,B 0,C 180,E1 -3940.147,E2 -3940.147} C_VEL
LIN {X 0,Y 538.018,Z 176.466,A -85,B 0,C 180,E1 -3943.299,E2 -3943.299} C_VEL
LIN {X 0,Y 538.053,Z 176.464,A -85,B 0,C 180,E1 -3945.63,E2 -3945.63} C_VEL
LIN {X 0,Y 538.078,Z 176.455,A -85,B 0,C 180,E1 -3948.701,E2 -3948.701} C_VEL
LIN {X 0,Y 538.08,Z 176.458,A -85,B 0,C 180,E1 -3951.739,E2 -3951.739} C_VEL
LIN {X 0,Y 538.152,Z 176.447,A -85,B 0,C 180,E1 -3954.755,E2 -3954.755} C_VEL
LIN {X 0,Y 538.15,Z 176.447,A -85,B 0,C 180,E1 -3957.755,E2 -3957.755} C_VEL
LIN {X 0,Y 538.175,Z 176.446,A -85,B 0,C 180,E1 -3960.748,E2 -3960.748} C_VEL
LIN {X 0,Y 538.126,Z 176.455,A -85,B 0,C 180,E1 -3962.995,E2 -3962.995} C_VEL
LIN {X 0,Y 538.101,Z 176.452,A -85,B 0,C 180,E1 -3965.998,E2 -3965.998} C_VEL
LIN {X 0,Y 538.07,Z 176.46,A -85,B 0,C 180,E1 -3968.261,E2 -3968.261} C_VEL
LIN {X 0,Y 538.073,Z 176.456,A -85,B 0,C 180,E1 -3971.598,E2 -3971.598} C_VEL
LIN {X 0,Y 538.047,Z 176.461,A -85,B 0,C 180,E1 -3974.858,E2 -3974.858} C_VEL
LIN {X 0,Y 538.024,Z 176.462,A -85,B 0,C 180,E1 -3977.533,E2 -3977.533} C_VEL
LIN {X 0,Y 538.02,Z 176.464,A -85,B 0,C 180,E1 -3980.652,E2 -3980.652} C_VEL
LIN {X 0,Y 537.994,Z 176.474,A -85,B 0,C 180,E1 -3983.878,E2 -3983.878} C_VEL
LIN {X 0,Y 537.97,Z 176.471,A -85,B 0,C 180,E1 -3986.371,E2 -3986.371} C_VEL
LIN {X 0,Y 537.98,Z 176.469,A -85,B 0,C 180,E1 -3988.926,E2 -3988.926} C_VEL
LIN {X 0,Y 537.997,Z 176.469,A -85,B 0,C 180,E1 -3991.887,E2 -3991.887} C_VEL
LIN {X 0,Y 537.989,Z 176.466,A -85,B 0,C 180,E1 -3994.617,E2 -3994.617} C_VEL
LIN {X 0,Y 537.989,Z 176.474,A -85,B 0,C 180,E1 -3997.17,E2 -3997.17} C_VEL
LIN {X 0,Y 537.999,Z 176.465,A -85,B 0,C 180,E1 -3999.799,E2 -3999.799} C_VEL
LIN {X 0,Y 537.991,Z 176.472,A -85,B 0,C 180,E1 -4002.789,E2 -4002.789} C_VEL
LIN {X 0,Y 537.996,Z 176.471,A -85,B 0,C 180,E1 -4005.139,E2 -4005.139} C_VEL
LIN {X 0,Y 538.023,Z 176.462,A -85,B 0,C 180,E1 -4008.228,E2 -4008.228} C_VEL
LIN {X 0,Y 538.008,Z 176.468,A -85,B 0,C 180,E1 -4011.171,E2 -4011.171} C_VEL
LIN {X 0,Y 537.99,Z 176.47,A -85,B 0,C 180,E1 -4014.09,E2 -4014.09} C_VEL
LIN {X 0,Y 538.026,Z 176.47,A -85,B 0,C 180,E1 -4016.729,E2 -4016.729} C_VEL
LIN {X 0,Y 538.047,Z 176.489,A -85,B 0,C 180,E1 -4018.563,E2 -4018.563} C_VEL
LIN {X 0,Y 540.428,Z 187.384,A -85,B 0,C 180,E1 -4020.611,E2 -4020.611} C_VEL
LIN {X 0,Y 540.045,Z 200.391,A -85,B 0,C 180,E1 -4022.722,E2 -4022.722} C_VEL
LIN {X 0,Y 539.539,Z 219.346,A -85,B 0,C 180,E1 -4025.65,E2 -4025.65} C_VEL
LIN {X 0,Y 539.124,Z 237.569,A -85,B 0,C 180,E1 -4028.393,E2 -4028.393} C_VEL
LIN {X 0,Y 538.732,Z 256.318,A -85,B 0,C 180,E1 -4031.164,E2 -4031.164} C_VEL
LIN {X 0,Y 538.396,Z 276.521,A -85,B 0,C 180,E1 -4034.091,E2 -4034.091} C_VEL
LIN {X 0,Y 538.183,Z 294.428,A -85,B 0,C 180,E1 -4036.623,E2 -4036.623} C_VEL
LIN {X 0,Y 539.232,Z 304.143,A -85,B 0,C 180,E1 -4036.817,E2 -4036.817} C_VEL
LIN {X 0,Y 539.026,Z 317.667,A -85,B 0,C 180,E1 -4037.171,E2 -4037.171} C_VEL
LIN {X 0,Y 538.834,Z 330.456,A -85,B 0,C 180,E1 -4037.669,E2 -4037.669} C_VEL
LIN {X 0,Y 538.651,Z 343.276,A -85,B 0,C 180,E1 -4038.343,E2 -4038.343} C_VEL
LIN {X 0,Y 538.435,Z 354.413,A -85,B 0,C 180,E1 -4039.091,E2 -4039.091} C_VEL
LIN {X 0,Y 538.245,Z 363.527,A -85,B 0,C 180,E1 -4039.848,E2 -4039.848} C_VEL
LIN {X 0,Y 538.029,Z 372.778,A -85,B 0,C 180,E1 -4040.793,E2 -4040.793} C_VEL
LIN {X 0,Y 537.85,Z 381.695,A -85,B 0,C 180,E1 -4041.926,E2 -4041.926} C_VEL
LIN {X 0,Y 537.727,Z 388.855,A -85,B 0,C 180,E1 -4043.057,E2 -4043.057} C_VEL
LIN {X 0,Y 537.676,Z 395.369,A -85,B 0,C 180,E1 -4044.375,E2 -4044.375} C_VEL
LIN {X 0,Y 537.557,Z 399.68,A -85,B 0,C 180,E1 -4045.502,E2 -4045.502} C_VEL
LIN {X 0,Y 537.591,Z 401.963,A -85,B 0,C 180,E1 -4046.253,E2 -4046.253} C_VEL
LIN {X 0,Y 537.551,Z 403.812,A -85,B 0,C 180,E1 -4047.003,E2 -4047.003} C_VEL
LIN {X 0,Y 537.451,Z 406.184,A -85,B 0,C 180,E1 -4048.502,E2 -4048.502} C_VEL
LIN {X 0,Y 537.442,Z 407,A -85,B 0,C 180,E1 -4050.001,E2 -4050.001} C_VEL
LIN {X 0,Y 537.451,Z 406.181,A -85,B 0,C 180,E1 -4051.5,E2 -4051.5} C_VEL
LIN {X 0,Y 537.551,Z 403.805,A -85,B 0,C 180,E1 -4052.999,E2 -4052.999} C_VEL
LIN {X 0,Y 537.604,Z 400.891,A -85,B 0,C 180,E1 -4054.124,E2 -4054.124} C_VEL
LIN {X 0,Y 537.588,Z 396.946,A -85,B 0,C 180,E1 -4055.252,E2 -4055.252} C_VEL
LIN {X 0,Y 537.652,Z 392.087,A -85,B 0,C 180,E1 -4056.334,E2 -4056.334} C_VEL
LIN {X 0,Y 537.792,Z 385.459,A -85,B 0,C 180,E1 -4057.51,E2 -4057.51} C_VEL
LIN {X 0,Y 537.97,Z 377.47,A -85,B 0,C 180,E1 -4058.641,E2 -4058.641} C_VEL
LIN {X 0,Y 538.119,Z 369.277,A -85,B 0,C 180,E1 -4059.586,E2 -4059.586} C_VEL
LIN {X 0,Y 538.366,Z 359.175,A -85,B 0,C 180,E1 -4060.531,E2 -4060.531} C_VEL
LIN {X 0,Y 538.54,Z 349.068,A -85,B 0,C 180,E1 -4061.289,E2 -4061.289} C_VEL
LIN {X 0,Y 538.715,Z 337.858,A -85,B 0,C 180,E1 -4061.965,E2 -4061.965} C_VEL
LIN {X 0,Y 538.94,Z 324.848,A -85,B 0,C 180,E1 -4062.57,E2 -4062.57} C_VEL
LIN {X 0,Y 539.107,Z 312.077,A -85,B 0,C 180,E1 -4062.997,E2 -4062.997} C_VEL
LIN {X 0,Y 539.056,Z 301.595,A -85,B 0,C 180,E1 -4063.237,E2 -4063.237} C_VEL
LIN {X 0,Y 538.184,Z 294.336,A -85,B 0,C 180,E1 -4063.379,E2 -4063.379} C_VEL
LIN {X 0,Y 538.453,Z 273.821,A -85,B 0,C 180,E1 -4066.298,E2 -4066.298} C_VEL
LIN {X 0,Y 538.737,Z 254.92,A -85,B 0,C 180,E1 -4069.035,E2 -4069.035} C_VEL
LIN {X 0,Y 539.082,Z 238.867,A -85,B 0,C 180,E1 -4071.411,E2 -4071.411} C_VEL
LIN {X 0,Y 539.514,Z 220.101,A -85,B 0,C 180,E1 -4074.236,E2 -4074.236} C_VEL
LIN {X 0,Y 540.007,Z 201.526,A -85,B 0,C 180,E1 -4077.099,E2 -4077.099} C_VEL
LIN {X 0,Y 540.473,Z 189.258,A -85,B 0,C 180,E1 -4079.073,E2 -4079.073} C_VEL
LIN {X 0,Y 540.196,Z 186.049,A -85,B 0,C 180,E1 -4079.63,E2 -4079.63} C_VEL
LIN {X 0,Y 538.039,Z 176.469,A -85,B 0,C 180,E1 -4081.445,E2 -4081.445} C_VEL
LIN {X 0,Y 538,Z 176.471,A -85,B 0,C 180,E1 -4084.175,E2 -4084.175} C_VEL
LIN {X 0,Y 538.003,Z 176.47,A -85,B 0,C 180,E1 -4087.169,E2 -4087.169} C_VEL
LIN {X 0,Y 538.014,Z 176.467,A -85,B 0,C 180,E1 -4089.799,E2 -4089.799} C_VEL
LIN {X 0,Y 538.024,Z 176.465,A -85,B 0,C 180,E1 -4092.786,E2 -4092.786} C_VEL
LIN {X 0,Y 538.023,Z 176.468,A -85,B 0,C 180,E1 -4095.927,E2 -4095.927} C_VEL
LIN {X 0,Y 538.035,Z 176.464,A -85,B 0,C 180,E1 -4098.227,E2 -4098.227} C_VEL
LIN {X 0,Y 538.013,Z 176.471,A -85,B 0,C 180,E1 -4101.169,E2 -4101.169} C_VEL
LIN {X 0,Y 537.971,Z 176.475,A -85,B 0,C 180,E1 -4104.093,E2 -4104.093} C_VEL
LIN {X 0,Y 537.987,Z 176.632,A -85,B 0,C 180,E1 -4105.937,E2 -4105.937} C_VEL
LIN {X 0,Y 537.991,Z 185.776,A -85,B 0,C 180,E1 -4108.497,E2 -4108.497} C_VEL
LIN {X 0,Y 538.009,Z 195.931,A -85,B 0,C 180,E1 -4111.523,E2 -4111.523} C_VEL
LIN {X 0,Y 538.056,Z 205.284,A -85,B 0,C 180,E1 -4114.466,E2 -4114.466} C_VEL
LIN {X 0,Y 538.006,Z 213.953,A -85,B 0,C 180,E1 -4117.334,E2 -4117.334} C_VEL
LIN {X 0,Y 537.967,Z 222.388,A -85,B 0,C 180,E1 -4120.155,E2 -4120.155} C_VEL
LIN {X 0,Y 537.876,Z 230.418,A -85,B 0,C 180,E1 -4122.909,E2 -4122.909} C_VEL
LIN {X 0,Y 537.821,Z 238.188,A -85,B 0,C 180,E1 -4125.624,E2 -4125.624} C_VEL
LIN {X 0,Y 537.749,Z 241.196,A -85,B 0,C 180,E1 -4126.707,E2 -4126.707} C_VEL
LIN {X 0,Y 539.216,Z 250.609,A -85,B 0,C 180,E1 -4126.959,E2 -4126.959} C_VEL
LIN {X 0,Y 539.082,Z 262.753,A -85,B 0,C 180,E1 -4127.339,E2 -4127.339} C_VEL
LIN {X 0,Y 538.849,Z 274.721,A -85,B 0,C 180,E1 -4127.859,E2 -4127.859} C_VEL
LIN {X 0,Y 538.666,Z 285.437,A -85,B 0,C 180,E1 -4128.465,E2 -4128.465} C_VEL
LIN {X 0,Y 538.415,Z 296.812,A -85,B 0,C 180,E1 -4129.28,E2 -4129.28} C_VEL
LIN {X 0,Y 538.198,Z 307.336,A -85,B 0,C 180,E1 -4130.226,E2 -4130.226} C_VEL
LIN {X 0,Y 538.015,Z 315.844,A -85,B 0,C 180,E1 -4131.171,E2 -4131.171} C_VEL
LIN {X 0,Y 537.818,Z 324.121,A -85,B 0,C 180,E1 -4132.303,E2 -4132.303} C_VEL
LIN {X 0,Y 537.682,Z 330.684,A -85,B 0,C 180,E1 -4133.413,E2 -4133.413} C_VEL
LIN {X 0,Y 537.675,Z 335.279,A -85,B 0,C 180,E1 -4134.374,E2 -4134.374} C_VEL
LIN {X 0,Y 537.566,Z 339.602,A -85,B 0,C 180,E1 -4135.501,E2 -4135.501} C_VEL
LIN {X 0,Y 537.592,Z 341.857,A -85,B 0,C 180,E1 -4136.252,E2 -4136.252} C_VEL
LIN {X 0,Y 537.489,Z 345.138,A -85,B 0,C 180,E1 -4137.752,E2 -4137.752} C_VEL
LIN {X 0,Y 537.443,Z 346.755,A -85,B 0,C 180,E1 -4139.251,E2 -4139.251} C_VEL
LIN {X 0,Y 537.442,Z 346.996,A -85,B 0,C 180,E1 -4140,E2 -4140} C_VEL
LIN {X 0,Y 537.442,Z 346.811,A -85,B 0,C 180,E1 -4140.749,E2 -4140.749} C_VEL
LIN {X 0,Y 537.489,Z 345.272,A -85,B 0,C 180,E1 -4142.248,E2 -4142.248} C_VEL
LIN {X 0,Y 537.552,Z 343.894,A -85,B 0,C 180,E1 -4142.998,E2 -4142.998} C_VEL
LIN {X 0,Y 537.604,Z 341.05,A -85,B 0,C 180,E1 -4144.123,E2 -4144.123} C_VEL
LIN {X 0,Y 537.587,Z 337.182,A -85,B 0,C 180,E1 -4145.251,E2 -4145.251} C_VEL
LIN {X 0,Y 537.681,Z 331.131,A -85,B 0,C 180,E1 -4146.587,E2 -4146.587} C_VEL
LIN {X 0,Y 537.817,Z 324.699,A -85,B 0,C 180,E1 -4147.698,E2 -4147.698} C_VEL
LIN {X 0,Y 537.958,Z 316.512,A -85,B 0,C 180,E1 -4148.83,E2 -4148.83} C_VEL
LIN {X 0,Y 538.145,Z 308.151,A -85,B 0,C 180,E1 -4149.775,E2 -4149.775} C_VEL
LIN {X 0,Y 538.388,Z 297.851,A -85,B 0,C 180,E1 -4150.72,E2 -4150.72} C_VEL
LIN {X 0,Y 538.596,Z 287.009,A -85,B 0,C 180,E1 -4151.52,E2 -4151.52} C_VEL
LIN {X 0,Y 538.818,Z 276.445,A -85,B 0,C 180,E1 -4152.141,E2 -4152.141} C_VEL
LIN {X 0,Y 539.061,Z 263.777,A -85,B 0,C 180,E1 -4152.71,E2 -4152.71} C_VEL
LIN {X 0,Y 539.225,Z 251.298,A -85,B 0,C 180,E1 -4153.113,E2 -4153.113} C_VEL
LIN {X 0,Y 537.913,Z 242.073,A -85,B 0,C 180,E1 -4153.346,E2 -4153.346} C_VEL
LIN {X 0,Y 537.699,Z 240.9,A -85,B 0,C 180,E1 -4153.391,E2 -4153.391} C_VEL
LIN {X 0,Y 537.792,Z 232.45,A -85,B 0,C 180,E1 -4156.318,E2 -4156.318} C_VEL
LIN {X 0,Y 537.908,Z 224.8,A -85,B 0,C 180,E1 -4159.065,E2 -4159.065} C_VEL
LIN {X 0,Y 538.007,Z 216.497,A -85,B 0,C 180,E1 -4161.954,E2 -4161.954} C_VEL
LIN {X 0,Y 538.079,Z 207.411,A -85,B 0,C 180,E1 -4165.119,E2 -4165.119} C_VEL
LIN {X 0,Y 538.151,Z 199.024,A -85,B 0,C 180,E1 -4168.044,E2 -4168.044} C_VEL
LIN {X 0,Y 538.291,Z 190.335,A -85,B 0,C 180,E1 -4171.092,E2 -4171.092} C_VEL
LIN {X 0,Y 538.269,Z 182.799,A -85,B 0,C 180,E1 -4173.704,E2 -4173.704} C_VEL
LIN {X 0,Y 538.288,Z 181.346,A -85,B 0,C 180,E1 -4174.211,E2 -4174.211} C_VEL
LIN {X 0,Y 537.608,Z 180.31,A -85,B 0,C 180,E1 -4174.611,E2 -4174.611} C_VEL
LIN {X 0,Y 534.671,Z 178.951,A -85,B 0,C 180,E1 -4175.241,E2 -4175.241} C_VEL
LIN {X 0,Y 531.688,Z 177.69,A -85,B 0,C 180,E1 -4175.886,E2 -4175.886} C_VEL
LIN {X 0,Y 530.963,Z 177.349,A -85,B 0,C 180,E1 -4176.31,E2 -4176.31} C_VEL
LIN {X 0,Y 530.99,Z 177.346,A -85,B 0,C 180,E1 -4179.443,E2 -4179.443} C_VEL
LIN {X 0,Y 530.964,Z 177.348,A -85,B 0,C 180,E1 -4182.458,E2 -4182.458} C_VEL
LIN {X 0,Y 530.98,Z 177.344,A -85,B 0,C 180,E1 -4185.622,E2 -4185.622} C_VEL
LIN {X 0,Y 530.999,Z 177.341,A -85,B 0,C 180,E1 -4188.564,E2 -4188.564} C_VEL
LIN {X 0,Y 530.957,Z 177.346,A -85,B 0,C 180,E1 -4191.528,E2 -4191.528} C_VEL
LIN {X 0,Y 530.937,Z 177.35,A -85,B 0,C 180,E1 -4194.378,E2 -4194.378} C_VEL
LIN {X 0,Y 530.972,Z 177.349,A -85,B 0,C 180,E1 -4197.133,E2 -4197.133} C_VEL
LIN {X 0,Y 530.923,Z 177.351,A -85,B 0,C 180,E1 -4199.799,E2 -4199.799} C_VEL
LIN {X 0,Y 530.852,Z 177.364,A -85,B 0,C 180,E1 -4200.901,E2 -4200.901} C_VEL
LIN {X 0,Y 530.821,Z 180.198,A -85,B 0,C 180,E1 -4203.246,E2 -4203.246} C_VEL
LIN {X 0,Y 530.738,Z 183.753,A -85,B 0,C 180,E1 -4206.022,E2 -4206.022} C_VEL
LIN {X 0,Y 530.674,Z 187.617,A -85,B 0,C 180,E1 -4209.048,E2 -4209.048} C_VEL
LIN {X 0,Y 530.617,Z 190.75,A -85,B 0,C 180,E1 -4211.464,E2 -4211.464} C_VEL
LIN {X 0,Y 530.572,Z 195.002,A -85,B 0,C 180,E1 -4214.637,E2 -4214.637} C_VEL
LIN {X 0,Y 530.55,Z 199.378,A -85,B 0,C 180,E1 -4217.763,E2 -4217.763} C_VEL
LIN {X 0,Y 530.496,Z 202.697,A -85,B 0,C 180,E1 -4220.082,E2 -4220.082} C_VEL
LIN {X 0,Y 530.527,Z 205.51,A -85,B 0,C 180,E1 -4222.028,E2 -4222.028} C_VEL
LIN {X 0,Y 531.398,Z 211.266,A -85,B 0,C 180,E1 -4222.256,E2 -4222.256} C_VEL
LIN {X 0,Y 531.354,Z 220.79,A -85,B 0,C 180,E1 -4222.724,E2 -4222.724} C_VEL
LIN {X 0,Y 531.244,Z 228.653,A -85,B 0,C 180,E1 -4223.262,E2 -4223.262} C_VEL
LIN {X 0,Y 531.068,Z 236.134,A -85,B 0,C 180,E1 -4223.922,E2 -4223.922} C_VEL
LIN {X 0,Y 531.026,Z 242.65,A -85,B 0,C 180,E1 -4224.683,E2 -4224.683} C_VEL
LIN {X 0,Y 530.907,Z 248.819,A -85,B 0,C 180,E1 -4225.634,E2 -4225.634} C_VEL
LIN {X 0,Y 530.855,Z 253.339,A -85,B 0,C 180,E1 -4226.584,E2 -4226.584} C_VEL
LIN {X 0,Y 530.657,Z 257.081,A -85,B 0,C 180,E1 -4227.722,E2 -4227.722} C_VEL
LIN {X 0,Y 530.649,Z 258.673,A -85,B 0,C 180,E1 -4228.481,E2 -4228.481} C_VEL
LIN {X 0,Y 530.614,Z 259.628,A -85,B 0,C 180,E1 -4229.24,E2 -4229.24} C_VEL
LIN {X 0,Y 530.604,Z 259.968,A -85,B 0,C 180,E1 -4229.999,E2 -4229.999} C_VEL
LIN {X 0,Y 530.613,Z 259.705,A -85,B 0,C 180,E1 -4230.758,E2 -4230.758} C_VEL
LIN {X 0,Y 530.581,Z 258.838,A -85,B 0,C 180,E1 -4231.517,E2 -4231.517} C_VEL
LIN {X 0,Y 530.738,Z 256.296,A -85,B 0,C 180,E1 -4232.655,E2 -4232.655} C_VEL
LIN {X 0,Y 530.813,Z 252.119,A -85,B 0,C 180,E1 -4233.795,E2 -4233.795} C_VEL
LIN {X 0,Y 530.968,Z 247.137,A -85,B 0,C 180,E1 -4234.744,E2 -4234.744} C_VEL
LIN {X 0,Y 531.046,Z 240.345,A -85,B 0,C 180,E1 -4235.695,E2 -4235.695} C_VEL
LIN {X 0,Y 531.087,Z 235.368,A -85,B 0,C 180,E1 -4236.241,E2 -4236.241} C_VEL
LIN {X 0,Y 531.254,Z 228.548,A -85,B 0,C 180,E1 -4236.837,E2 -4236.837} C_VEL
LIN {X 0,Y 531.322,Z 220.118,A -85,B 0,C 180,E1 -4237.409,E2 -4237.409} C_VEL
LIN {X 0,Y 531.435,Z 211.185,A -85,B 0,C 180,E1 -4237.837,E2 -4237.837} C_VEL
LIN {X 0,Y 530.515,Z 205.452,A -85,B 0,C 180,E1 -4238.09,E2 -4238.09} C_VEL
LIN {X 0,Y 530.604,Z 200.608,A -85,B 0,C 180,E1 -4241.459,E2 -4241.459} C_VEL
LIN {X 0,Y 530.577,Z 195.958,A -85,B 0,C 180,E1 -4244.77,E2 -4244.77} C_VEL
LIN {X 0,Y 530.604,Z 191.934,A -85,B 0,C 180,E1 -4247.735,E2 -4247.735} C_VEL
LIN {X 0,Y 530.665,Z 188.782,A -85,B 0,C 180,E1 -4250.14,E2 -4250.14} C_VEL
LIN {X 0,Y 530.699,Z 185.676,A -85,B 0,C 180,E1 -4252.583,E2 -4252.583} C_VEL
LIN {X 0,Y 530.761,Z 182.514,A -85,B 0,C 180,E1 -4255.069,E2 -4255.069} C_VEL
LIN {X 0,Y 530.8,Z 179.209,A -85,B 0,C 180,E1 -4257.606,E2 -4257.606} C_VEL
LIN {X 0,Y 530.838,Z 177.366,A -85,B 0,C 180,E1 -4259.096,E2 -4259.096} C_VEL
LIN {X 0,Y 530.942,Z 177.347,A -85,B 0,C 180,E1 -4261.079,E2 -4261.079} C_VEL
LIN {X 0,Y 530.985,Z 177.345,A -85,B 0,C 180,E1 -4263.771,E2 -4263.771} C_VEL
LIN {X 0,Y 530.961,Z 177.342,A -85,B 0,C 180,E1 -4266.556,E2 -4266.556} C_VEL
LIN {X 0,Y 530.975,Z 177.342,A -85,B 0,C 180,E1 -4269.853,E2 -4269.853} C_VEL
LIN {X 0,Y 530.975,Z 177.341,A -85,B 0,C 180,E1 -4272.455,E2 -4272.455} C_VEL
LIN {X 0,Y 530.979,Z 177.341,A -85,B 0,C 180,E1 -4275.62,E2 -4275.62} C_VEL
LIN {X 0,Y 530.993,Z 177.342,A -85,B 0,C 180,E1 -4278.564,E2 -4278.564} C_VEL
LIN {X 0,Y 530.952,Z 177.343,A -85,B 0,C 180,E1 -4281.529,E2 -4281.529} C_VEL
LIN {X 0,Y 530.975,Z 177.345,A -85,B 0,C 180,E1 -4284.381,E2 -4284.381} C_VEL
LIN {X 0,Y 530.967,Z 177.342,A -85,B 0,C 180,E1 -4287.133,E2 -4287.133} C_VEL
LIN {X 0,Y 530.977,Z 177.341,A -85,B 0,C 180,E1 -4289.803,E2 -4289.803} C_VEL
LIN {X 0,Y 531.008,Z 177.341,A -85,B 0,C 180,E1 -4292.465,E2 -4292.465} C_VEL
LIN {X 0,Y 530.998,Z 177.335,A -85,B 0,C 180,E1 -4294.942,E2 -4294.942} C_VEL
LIN {X 0,Y 530.962,Z 177.345,A -85,B 0,C 180,E1 -4298.246,E2 -4298.246} C_VEL
LIN {X 0,Y 530.987,Z 177.338,A -85,B 0,C 180,E1 -4300.677,E2 -4300.677} C_VEL
LIN {X 0,Y 530.983,Z 177.34,A -85,B 0,C 180,E1 -4303.071,E2 -4303.071} C_VEL
LIN {X 0,Y 531.008,Z 177.339,A -85,B 0,C 180,E1 -4305.435,E2 -4305.435} C_VEL
LIN {X 0,Y 531.035,Z 177.332,A -85,B 0,C 180,E1 -4308.55,E2 -4308.55} C_VEL
LIN {X 0,Y 531.049,Z 177.335,A -85,B 0,C 180,E1 -4311.629,E2 -4311.629} C_VEL
LIN {X 0,Y 531.111,Z 177.323,A -85,B 0,C 180,E1 -4314.685,E2 -4314.685} C_VEL
LIN {X 0,Y 531.123,Z 177.322,A -85,B 0,C 180,E1 -4317.725,E2 -4317.725} C_VEL
LIN {X 0,Y 531.145,Z 177.322,A -85,B 0,C 180,E1 -4320.758,E2 -4320.758} C_VEL
LIN {X 0,Y 531.092,Z 177.33,A -85,B 0,C 180,E1 -4323.034,E2 -4323.034} C_VEL
LIN {X 0,Y 531.058,Z 177.33,A -85,B 0,C 180,E1 -4326.077,E2 -4326.077} C_VEL
LIN {X 0,Y 531.04,Z 177.338,A -85,B 0,C 180,E1 -4328.371,E2 -4328.371} C_VEL
LIN {X 0,Y 531.036,Z 177.333,A -85,B 0,C 180,E1 -4331.671,E2 -4331.671} C_VEL
LIN {X 0,Y 531.019,Z 177.336,A -85,B 0,C 180,E1 -4334.956,E2 -4334.956} C_VEL
LIN {X 0,Y 530.967,Z 177.343,A -85,B 0,C 180,E1 -4337.724,E2 -4337.724} C_VEL
LIN {X 0,Y 531.012,Z 177.344,A -85,B 0,C 180,E1 -4340.128,E2 -4340.128} C_VEL
LIN {X 0,Y 530.928,Z 177.348,A -85,B 0,C 180,E1 -4342.574,E2 -4342.574} C_VEL
LIN {X 0,Y 530.936,Z 177.346,A -85,B 0,C 180,E1 -4345.061,E2 -4345.061} C_VEL
LIN {X 0,Y 530.938,Z 177.353,A -85,B 0,C 180,E1 -4347.6,E2 -4347.6} C_VEL
LIN {X 0,Y 530.947,Z 177.344,A -85,B 0,C 180,E1 -4350.643,E2 -4350.643} C_VEL
LIN {X 0,Y 530.952,Z 177.346,A -85,B 0,C 180,E1 -4353.775,E2 -4353.775} C_VEL
LIN {X 0,Y 530.939,Z 177.346,A -85,B 0,C 180,E1 -4356.56,E2 -4356.56} C_VEL
LIN {X 0,Y 530.96,Z 177.345,A -85,B 0,C 180,E1 -4359.446,E2 -4359.446} C_VEL
LIN {X 0,Y 530.955,Z 177.345,A -85,B 0,C 180,E1 -4362.459,E2 -4362.459} C_VEL
LIN {X 0,Y 530.968,Z 177.342,A -85,B 0,C 180,E1 -4365.623,E2 -4365.623} C_VEL
LIN {X 0,Y 530.986,Z 177.342,A -85,B 0,C 180,E1 -4368.565,E2 -4368.565} C_VEL
LIN {X 0,Y 530.951,Z 177.345,A -85,B 0,C 180,E1 -4371.53,E2 -4371.53} C_VEL
LIN {X 0,Y 530.95,Z 177.352,A -85,B 0,C 180,E1 -4374.381,E2 -4374.381} C_VEL
LIN {X 0,Y 530.963,Z 177.347,A -85,B 0,C 180,E1 -4377.135,E2 -4377.135} C_VEL
LIN {X 0,Y 530.996,Z 177.494,A -85,B 0,C 180,E1 -4378.286,E2 -4378.286} C_VEL
LIN {X 0,Y 533.614,Z 189.175,A -85,B 0,C 180,E1 -4380.53,E2 -4380.53} C_VEL
LIN {X 0,Y 533.188,Z 201.256,A -85,B 0,C 180,E1 -4382.528,E2 -4382.528} C_VEL
LIN {X 0,Y 532.654,Z 218.199,A -85,B 0,C 180,E1 -4385.193,E2 -4385.193} C_VEL
LIN {X 0,Y 532.203,Z 237.265,A -85,B 0,C 180,E1 -4388.109,E2 -4388.109} C_VEL
LIN {X 0,Y 531.74,Z 255.851,A -85,B 0,C 180,E1 -4390.907,E2 -4390.907} C_VEL
LIN {X 0,Y 531.361,Z 275.911,A -85,B 0,C 180,E1 -4393.875,E2 -4393.875} C_VEL
LIN {X 0,Y 531.12,Z 293.878,A -85,B 0,C 180,E1 -4396.49,E2 -4396.49} C_VEL
LIN {X 0,Y 532.224,Z 304.828,A -85,B 0,C 180,E1 -4396.713,E2 -4396.713} C_VEL
LIN {X 0,Y 532.012,Z 317.709,A -85,B 0,C 180,E1 -4397.072,E2 -4397.072} C_VEL
LIN {X 0,Y 531.771,Z 330.662,A -85,B 0,C 180,E1 -4397.599,E2 -4397.599} C_VEL
LIN {X 0,Y 531.598,Z 342.595,A -85,B 0,C 180,E1 -4398.245,E2 -4398.245} C_VEL
LIN {X 0,Y 531.347,Z 354.118,A -85,B 0,C 180,E1 -4399.04,E2 -4399.04} C_VEL
LIN {X 0,Y 531.142,Z 364.172,A -85,B 0,C 180,E1 -4399.904,E2 -4399.904} C_VEL
LIN {X 0,Y 530.95,Z 373.317,A -85,B 0,C 180,E1 -4400.862,E2 -4400.862} C_VEL
LIN {X 0,Y 530.754,Z 382.228,A -85,B 0,C 180,E1 -4402.009,E2 -4402.009} C_VEL
LIN {X 0,Y 530.635,Z 389.342,A -85,B 0,C 180,E1 -4403.155,E2 -4403.155} C_VEL
LIN {X 0,Y 530.59,Z 395.034,A -85,B 0,C 180,E1 -4404.3,E2 -4404.3} C_VEL
LIN {X 0,Y 530.454,Z 399.474,A -85,B 0,C 180,E1 -4405.442,E2 -4405.442} C_VEL
LIN {X 0,Y 530.516,Z 401.829,A -85,B 0,C 180,E1 -4406.203,E2 -4406.203} C_VEL
